DATA_BLOCK "Drives --> Plc"	// DB 1
TITLE = DRIVE --> PLC DATA BLOCK
AUTHOR : Milesi
VERSION : 0.1
  STRUCT
   TRVERSE_STATUS_W1 : STRUCT
    DB1_DBX0_0 : BOOL ;	//Setpoint/actual value deviation detected
    DB1_DBX0_1 : BOOL ;	//PZD control requests
    DB1_DBX0_2 : BOOL ;	//Actual value>=Comparsion setpoint
    DB1_DBX0_3 : BOOL ;	//Undervoltage fault
    DB1_DBX0_4 : BOOL ;	//Request to energize main contactor
    DB1_DBX0_5 : BOOL ;	//Ramp-function generetor active
    DB1_DBX0_6 : BOOL ;	//Positive speed setpoint
    DB1_DBX0_7 : BOOL ;	//Kinetic buffering/flexible response active
    DB1_DBX1_0 : BOOL ;	//Ready to switch on
    DB1_DBX1_1 : BOOL ;	//Ready to operate
    DB1_DBX1_2 : BOOL ;	//Run
    DB1_DBX1_3 : BOOL ;	//Fault is active
    DB1_DBX1_4 : BOOL ;	//OFF2 applied
    DB1_DBX1_5 : BOOL ;	//OFF3 applied
    DB1_DBX1_6 : BOOL ;	//Switch on inhibit
    DB1_DBX1_7 : BOOL ;	//Alarm is active
   END_STRUCT ;
   TRAVERSE_STATUS_W2 : STRUCT
    DB1_DBX2_0 : BOOL ;	//Power section overtemperature alarm active
    DB1_DBX2_1 : BOOL ;	//Motor overtemperature alarm active
    DB1_DBX2_2 : BOOL ;	//Motor overtemperature fault active
    DB1_DBX2_3 : BOOL ;	//Spare
    DB1_DBX2_4 : BOOL ;	//Motor locked fault active
    DB1_DBX2_5 : BOOL ;	//Spare
    DB1_DBX2_6 : BOOL ;	//Spare
    DB1_DBX2_7 : BOOL ;	//Spare
    DB1_DBX3_0 : BOOL ;	//Spare
    DB1_DBX3_1 : BOOL ;	//Spare
    DB1_DBX3_2 : BOOL ;	//Overspeed
    DB1_DBX3_3 : BOOL ;	//External fault 1 active
    DB1_DBX3_4 : BOOL ;	//External fault 2 active
    DB1_DBX3_5 : BOOL ;	//External alarm active
    DB1_DBX3_6 : BOOL ;	//Power section overload alarm active
    DB1_DBX3_7 : BOOL ;	//Power section overtemperature fault active
   END_STRUCT ;
   DB1_DBW4 : INT ;
   DB1_DBW6 : INT ;	//Motor speed
   DB1_DBW8 : INT ;	//Motor current
   DB1_DBW10 : INT ;	//Motor voltage
   DB1_DBW12 : INT ;
   DB1_DBW14 : INT ;
   DB1_DBW16 : INT ;
   DB1_DBW18 : INT ;
   DB1_DBW20 : INT ;
   DB1_DBW22 : INT ;
   DB1_DBW24 : INT ;
   DB1_DBW26 : INT ;
   DB1_DBW28 : INT ;
   DB1_DBW30 : INT ;
   DB1_DBW32 : INT ;
   DB1_DBW34 : INT ;
   DB1_DBW36 : INT ;
   DB1_DBW38 : INT ;
   BOBBIN_STATUS_W1 : STRUCT
    DB1_DBX40_0 : BOOL ;	//Setpoint/actual value deviation detected
    DB1_DBX40_1 : BOOL ;	//PZD control requests
    DB1_DBX40_2 : BOOL ;	//Actual value>=Comparsion setpoint
    DB1_DBX40_3 : BOOL ;	//Undervoltage fault
    DB1_DBX40_4 : BOOL ;	//Request to energize main contactor
    DB1_DBX40_5 : BOOL ;	//Ramp-function generetor active
    DB1_DBX40_6 : BOOL ;	//Positive speed setpoint
    DB1_DBX40_7 : BOOL ;	//Kinetic buffering/flexible response active
    DB1_DBX41_0 : BOOL ;	//Ready to switch on
    DB1_DBX41_1 : BOOL ;	//Ready to operate
    DB1_DBX41_2 : BOOL ;	//Run
    DB1_DBX41_3 : BOOL ;	//Fault is active
    DB1_DBX41_4 : BOOL ;	//OFF2 applied
    DB1_DBX41_5 : BOOL ;	//OFF3 applied
    DB1_DBX41_6 : BOOL ;	//Switch on inhibit
    DB1_DBX41_7 : BOOL ;	//Alarm is active
   END_STRUCT ;
   BOBBIN_STATUS_W2 : STRUCT
    DB1_DBX42_0 : BOOL ;	//Power section overtemperature alarm active
    DB1_DBX42_1 : BOOL ;	//Motor overtemperature alarm active
    DB1_DBX42_2 : BOOL ;	//Motor overtemperature fault active
    DB1_DBX42_3 : BOOL ;	//Spare
    DB1_DBX42_4 : BOOL ;	//Motor locked fault active
    DB1_DBX42_5 : BOOL ;	//Spare
    DB1_DBX42_6 : BOOL ;	//Spare
    DB1_DBX42_7 : BOOL ;	//Spare
    DB1_DBX43_0 : BOOL ;	//Spare
    DB1_DBX43_1 : BOOL ;	//Spare
    DB1_DBX43_2 : BOOL ;	//Overspeed
    DB1_DBX43_3 : BOOL ;	//External fault 1 active
    DB1_DBX43_4 : BOOL ;	//External fault 2 active
    DB1_DBX43_5 : BOOL ;	//External alarm active
    DB1_DBX43_6 : BOOL ;	//Power section overload alarm active
    DB1_DBX43_7 : BOOL ;	//Power section overtemperature fault active
   END_STRUCT ;
   DB1_DBW44 : INT ;
   DB1_DBW46 : INT ;	//Motor speed
   DB1_DBW48 : INT ;	//Motor current
   DB1_DBW50 : INT ;	//Motor voltage
   DB1_DBW52 : INT ;
   DB1_DBW54 : INT ;
   DB1_DBW56 : INT ;
   DB1_DBW58 : INT ;
   DB1_DBW60 : INT ;
   DB1_DBW62 : INT ;
   DB1_DBW64 : INT ;
   DB1_DBW66 : INT ;
   DB1_DBW68 : INT ;
   DB1_DBW70 : INT ;
   DB1_DBW72 : INT ;
   DB1_DBW74 : INT ;
   DB1_DBW76 : INT ;
   DB1_DBW78 : INT ;
   CAPSTAN_STATUS_W1 : STRUCT
    DB1_DBX80_0 : BOOL ;	//Setpoint/actual value deviation detected
    DB1_DBX80_1 : BOOL ;	//PZD control requests
    DB1_DBX80_2 : BOOL ;	//Actual value>=Comparsion setpoint
    DB1_DBX80_3 : BOOL ;	//Undervoltage fault
    DB1_DBX80_4 : BOOL ;	//Request to energize main contactor
    DB1_DBX80_5 : BOOL ;	//Ramp-function generetor active
    DB1_DBX80_6 : BOOL ;	//Positive speed setpoint
    DB1_DBX80_7 : BOOL ;	//Kinetic buffering/flexible response active
    DB1_DBX81_0 : BOOL ;	//Ready to switch on
    DB1_DBX81_1 : BOOL ;	//Ready to operate
    DB1_DBX81_2 : BOOL ;	//Run
    DB1_DBX81_3 : BOOL ;	//Fault is active
    DB1_DBX81_4 : BOOL ;	//OFF2 applied
    DB1_DBX81_5 : BOOL ;	//OFF3 applied
    DB1_DBX81_6 : BOOL ;	//Switch on inhibit
    DB1_DBX81_7 : BOOL ;	//Alarm is active
   END_STRUCT ;
   CAPSTAN_STATUS_W2 : STRUCT
    DB1_DBX82_0 : BOOL ;	//Power section overtemperature alarm active
    DB1_DBX82_1 : BOOL ;	//Motor overtemperature alarm active
    DB1_DBX82_2 : BOOL ;	//Motor overtemperature fault active
    DB1_DBX82_3 : BOOL ;	//Spare
    DB1_DBX82_4 : BOOL ;	//Motor locked fault active
    DB1_DBX82_5 : BOOL ;	//Spare
    DB1_DBX82_6 : BOOL ;	//Spare
    DB1_DBX82_7 : BOOL ;	//Spare
    DB1_DBX83_0 : BOOL ;	//Spare
    DB1_DBX83_1 : BOOL ;	//Spare
    DB1_DBX83_2 : BOOL ;	//Overspeed
    DB1_DBX83_3 : BOOL ;	//External fault 1 active
    DB1_DBX83_4 : BOOL ;	//External fault 2 active
    DB1_DBX83_5 : BOOL ;	//External alarm active
    DB1_DBX83_6 : BOOL ;	//Power section overload alarm active
    DB1_DBX83_7 : BOOL ;	//Power section overtemperature fault active
   END_STRUCT ;
   DB1_DBW84 : INT ;
   DB1_DBW86 : INT ;	//Motor speed
   DB1_DBW88 : INT ;	//Motor current
   DB1_DBW90 : INT ;	//Motor voltage
   DB1_DBW92 : INT ;
   DB1_DBW94 : INT ;
   DB1_DBW96 : INT ;
   DB1_DBW98 : INT ;
   DB1_DBW100 : INT ;
   DB1_DBW102 : INT ;
   DB1_DBW104 : INT ;
   DB1_DBW106 : INT ;
   DB1_DBW108 : INT ;
   DB1_DBW110 : INT ;
   DB1_DBW112 : INT ;
   DB1_DBW114 : INT ;
   DB1_DBW116 : INT ;
   DB1_DBW118 : INT ;
   CAGE_24_PREF_STATUS_W1 : STRUCT
    DB1_DBX120_0 : BOOL ;	//Setpoint/actual value deviation detected
    DB1_DBX120_1 : BOOL ;	//PZD control requests
    DB1_DBX120_2 : BOOL ;	//Actual value>=Comparsion setpoint
    DB1_DBX120_3 : BOOL ;	//Undervoltage fault
    DB1_DBX120_4 : BOOL ;	//Request to energize main contactor
    DB1_DBX120_5 : BOOL ;	//Ramp-function generetor active
    DB1_DBX120_6 : BOOL ;	//Positive speed setpoint
    DB1_DBX120_7 : BOOL ;	//Kinetic buffering/flexible response active
    DB1_DBX121_0 : BOOL ;	//Ready to switch on
    DB1_DBX121_1 : BOOL ;	//Ready to operate
    DB1_DBX121_2 : BOOL ;	//Run
    DB1_DBX121_3 : BOOL ;	//Fault is active
    DB1_DBX121_4 : BOOL ;	//OFF2 applied
    DB1_DBX121_5 : BOOL ;	//OFF3 applied
    DB1_DBX121_6 : BOOL ;	//Switch on inhibit
    DB1_DBX121_7 : BOOL ;	//Alarm is active
   END_STRUCT ;
   CAGE_24_PREF_STATUS_W2 : STRUCT
    DB1_DBX122_0 : BOOL ;	//Power section overtemperature alarm active
    DB1_DBX122_1 : BOOL ;	//Motor overtemperature alarm active
    DB1_DBX122_2 : BOOL ;	//Motor overtemperature fault active
    DB1_DBX122_3 : BOOL ;	//Spare
    DB1_DBX122_4 : BOOL ;	//Motor locked fault active
    DB1_DBX122_5 : BOOL ;	//Spare
    DB1_DBX122_6 : BOOL ;	//Spare
    DB1_DBX122_7 : BOOL ;	//Spare
    DB1_DBX123_0 : BOOL ;	//Spare
    DB1_DBX123_1 : BOOL ;	//Spare
    DB1_DBX123_2 : BOOL ;	//Overspeed
    DB1_DBX123_3 : BOOL ;	//External fault 1 active
    DB1_DBX123_4 : BOOL ;	//External fault 2 active
    DB1_DBX123_5 : BOOL ;	//External alarm active
    DB1_DBX123_6 : BOOL ;	//Power section overload alarm active
    DB1_DBX123_7 : BOOL ;	//Power section overtemperature fault active
   END_STRUCT ;
   DB1_DBW124 : INT ;
   DB1_DBW126 : INT ;	//Motor speed
   DB1_DBW128 : INT ;	//Motor current
   DB1_DBW130 : INT ;	//Motor voltage
   DB1_DBW132 : INT ;
   DB1_DBW134 : INT ;
   DB1_DBW136 : INT ;
   DB1_DBW138 : INT ;
   DB1_DBW140 : INT ;
   DB1_DBW142 : INT ;
   DB1_DBW144 : INT ;
   DB1_DBW146 : INT ;
   DB1_DBW148 : INT ;
   DB1_DBW150 : INT ;
   DB1_DBW152 : INT ;
   DB1_DBW154 : INT ;
   DB1_DBW156 : INT ;
   DB1_DBW158 : INT ;
   CAGE_24_STATUS_W1 : STRUCT
    DB1_DBX160_0 : BOOL ;	//Setpoint/actual value deviation detected
    DB1_DBX160_1 : BOOL ;	//PZD control requests
    DB1_DBX160_2 : BOOL ;	//Actual value>=Comparsion setpoint
    DB1_DBX160_3 : BOOL ;	//Undervoltage fault
    DB1_DBX160_4 : BOOL ;	//Request to energize main contactor
    DB1_DBX160_5 : BOOL ;	//Ramp-function generetor active
    DB1_DBX160_6 : BOOL ;	//Positive speed setpoint
    DB1_DBX160_7 : BOOL ;	//Kinetic buffering/flexible response active
    DB1_DBX161_0 : BOOL ;	//Ready to switch on
    DB1_DBX161_1 : BOOL ;	//Ready to operate
    DB1_DBX161_2 : BOOL ;	//Run
    DB1_DBX161_3 : BOOL ;	//Fault is active
    DB1_DBX161_4 : BOOL ;	//OFF2 applied
    DB1_DBX161_5 : BOOL ;	//OFF3 applied
    DB1_DBX161_6 : BOOL ;	//Switch on inhibit
    DB1_DBX161_7 : BOOL ;	//Alarm is active
   END_STRUCT ;
   CAGE_24_STATUS_W2 : STRUCT
    DB1_DBX162_0 : BOOL ;	//Power section overtemperature alarm active
    DB1_DBX162_1 : BOOL ;	//Motor overtemperature alarm active
    DB1_DBX162_2 : BOOL ;	//Motor overtemperature fault active
    DB1_DBX162_3 : BOOL ;	//Spare
    DB1_DBX162_4 : BOOL ;	//Motor locked fault active
    DB1_DBX162_5 : BOOL ;	//Spare
    DB1_DBX162_6 : BOOL ;	//Spare
    DB1_DBX162_7 : BOOL ;	//Spare
    DB1_DBX163_0 : BOOL ;	//Spare
    DB1_DBX163_1 : BOOL ;	//Spare
    DB1_DBX163_2 : BOOL ;	//Overspeed
    DB1_DBX163_3 : BOOL ;	//External fault 1 active
    DB1_DBX163_4 : BOOL ;	//External fault 2 active
    DB1_DBX163_5 : BOOL ;	//External alarm active
    DB1_DBX163_6 : BOOL ;	//Power section overload alarm active
    DB1_DBX163_7 : BOOL ;	//Power section overtemperature fault active
   END_STRUCT ;
   DB1_DBW1641 : INT ;
   DB1_DBW1661 : INT ;	//Motor speed
   DB1_DBW1681 : INT ;	//Motor current
   DB1_DBW1701 : INT ;	//Motor voltage
   DB1_DBW1721 : INT ;
   DB1_DBW1741 : INT ;
   DB1_DBW1761 : INT ;
   DB1_DBW1781 : INT ;
   DB1_DBW1801 : INT ;
   DB1_DBW1821 : INT ;
   DB1_DBW1841 : INT ;
   DB1_DBW1861 : INT ;
   DB1_DBW1881 : INT ;
   DB1_DBW1901 : INT ;
   DB1_DBW1921 : INT ;
   DB1_DBW1941 : INT ;
   DB1_DBW1961 : INT ;
   DB1_DBW1981 : INT ;
   CAGE_18_PREF_STATUS_W1 : STRUCT
    DB1_DBX200_0 : BOOL ;	//Setpoint/actual value deviation detected
    DB1_DBX200_1 : BOOL ;	//PZD control requests
    DB1_DBX200_2 : BOOL ;	//Actual value>=Comparsion setpoint
    DB1_DBX200_3 : BOOL ;	//Undervoltage fault
    DB1_DBX200_4 : BOOL ;	//Request to energize main contactor
    DB1_DBX200_5 : BOOL ;	//Ramp-function generetor active
    DB1_DBX200_6 : BOOL ;	//Positive speed setpoint
    DB1_DBX200_7 : BOOL ;	//Kinetic buffering/flexible response active
    DB1_DBX201_0 : BOOL ;	//Ready to switch on
    DB1_DBX201_1 : BOOL ;	//Ready to operate
    DB1_DBX201_2 : BOOL ;	//Run
    DB1_DBX201_3 : BOOL ;	//Fault is active
    DB1_DBX201_4 : BOOL ;	//OFF2 applied
    DB1_DBX201_5 : BOOL ;	//OFF3 applied
    DB1_DBX201_6 : BOOL ;	//Switch on inhibit
    DB1_DBX201_7 : BOOL ;	//Alarm is active
   END_STRUCT ;
   CAGE_18_PREF_STATUS_W2 : STRUCT
    DB1_DBX202_0 : BOOL ;	//Power section overtemperature alarm active
    DB1_DBX202_1 : BOOL ;	//Motor overtemperature alarm active
    DB1_DBX202_2 : BOOL ;	//Motor overtemperature fault active
    DB1_DBX202_3 : BOOL ;	//Spare
    DB1_DBX202_4 : BOOL ;	//Motor locked fault active
    DB1_DBX202_5 : BOOL ;	//Spare
    DB1_DBX202_6 : BOOL ;	//Spare
    DB1_DBX202_7 : BOOL ;	//Spare
    DB1_DBX203_0 : BOOL ;	//Spare
    DB1_DBX203_1 : BOOL ;	//Spare
    DB1_DBX203_2 : BOOL ;	//Overspeed
    DB1_DBX203_3 : BOOL ;	//External fault 1 active
    DB1_DBX203_4 : BOOL ;	//External fault 2 active
    DB1_DBX203_5 : BOOL ;	//External alarm active
    DB1_DBX203_6 : BOOL ;	//Power section overload alarm active
    DB1_DBX203_7 : BOOL ;	//Power section overtemperature fault active
   END_STRUCT ;
   DB1_DBW204 : INT ;
   DB1_DBW206 : INT ;	//Motor speed
   DB1_DBW208 : INT ;	//Motor current
   DB1_DBW210 : INT ;	//Motor voltage
   DB1_DBW212 : INT ;
   DB1_DBW214 : INT ;
   DB1_DBW216 : INT ;
   DB1_DBW218 : INT ;
   DB1_DBW220 : INT ;
   DB1_DBW222 : INT ;
   DB1_DBW224 : INT ;
   DB1_DBW226 : INT ;
   DB1_DBW228 : INT ;
   DB1_DBW230 : INT ;
   DB1_DBW232 : INT ;
   DB1_DBW234 : INT ;
   DB1_DBW236 : INT ;
   DB1_DBW238 : INT ;
   CAGE_18_STATUS_W1 : STRUCT
    DB1_DBX240_0 : BOOL ;	//Setpoint/actual value deviation detected
    DB1_DBX240_1 : BOOL ;	//PZD control requests
    DB1_DBX240_2 : BOOL ;	//Actual value>=Comparsion setpoint
    DB1_DBX240_3 : BOOL ;	//Undervoltage fault
    DB1_DBX240_4 : BOOL ;	//Request to energize main contactor
    DB1_DBX240_5 : BOOL ;	//Ramp-function generetor active
    DB1_DBX240_6 : BOOL ;	//Positive speed setpoint
    DB1_DBX240_7 : BOOL ;	//Kinetic buffering/flexible response active
    DB1_DBX241_0 : BOOL ;	//Ready to switch on
    DB1_DBX241_1 : BOOL ;	//Ready to operate
    DB1_DBX241_2 : BOOL ;	//Run
    DB1_DBX241_3 : BOOL ;	//Fault is active
    DB1_DBX241_4 : BOOL ;	//OFF2 applied
    DB1_DBX241_5 : BOOL ;	//OFF3 applied
    DB1_DBX241_6 : BOOL ;	//Switch on inhibit
    DB1_DBX241_7 : BOOL ;	//Alarm is active
   END_STRUCT ;
   CAGE_18_STATUS_W2 : STRUCT
    DB1_DBX242_0 : BOOL ;	//Power section overtemperature alarm active
    DB1_DBX242_1 : BOOL ;	//Motor overtemperature alarm active
    DB1_DBX242_2 : BOOL ;	//Motor overtemperature fault active
    DB1_DBX242_3 : BOOL ;	//Spare
    DB1_DBX242_4 : BOOL ;	//Motor locked fault active
    DB1_DBX242_5 : BOOL ;	//Spare
    DB1_DBX242_6 : BOOL ;	//Spare
    DB1_DBX242_7 : BOOL ;	//Spare
    DB1_DBX243_0 : BOOL ;	//Spare
    DB1_DBX243_1 : BOOL ;	//Spare
    DB1_DBX243_2 : BOOL ;	//Overspeed
    DB1_DBX243_3 : BOOL ;	//External fault 1 active
    DB1_DBX243_4 : BOOL ;	//External fault 2 active
    DB1_DBX243_5 : BOOL ;	//External alarm active
    DB1_DBX243_6 : BOOL ;	//Power section overload alarm active
    DB1_DBX243_7 : BOOL ;	//Power section overtemperature fault active
   END_STRUCT ;
   DB1_DBW244 : INT ;
   DB1_DBW246 : INT ;	//Motor speed
   DB1_DBW248 : INT ;	//Motor current
   DB1_DBW250 : INT ;	//Motor voltage
   DB1_DBW252 : INT ;
   DB1_DBW254 : INT ;
   DB1_DBW256 : INT ;
   DB1_DBW258 : INT ;
   DB1_DBW260 : INT ;
   DB1_DBW262 : INT ;
   DB1_DBW264 : INT ;
   DB1_DBW266 : INT ;
   DB1_DBW268 : INT ;
   DB1_DBW270 : INT ;
   DB1_DBW272 : INT ;
   DB1_DBW274 : INT ;
   DB1_DBW276 : INT ;
   DB1_DBW278 : INT ;
   CAGE_12_PREF_STATUS_W1 : STRUCT
    DB1_DBX280_0 : BOOL ;	//Setpoint/actual value deviation detected
    DB1_DBX280_1 : BOOL ;	//PZD control requests
    DB1_DBX280_2 : BOOL ;	//Actual value>=Comparsion setpoint
    DB1_DBX280_3 : BOOL ;	//Undervoltage fault
    DB1_DBX280_4 : BOOL ;	//Request to energize main contactor
    DB1_DBX280_5 : BOOL ;	//Ramp-function generetor active
    DB1_DBX280_6 : BOOL ;	//Positive speed setpoint
    DB1_DBX280_7 : BOOL ;	//Kinetic buffering/flexible response active
    DB1_DBX281_0 : BOOL ;	//Ready to switch on
    DB1_DBX281_1 : BOOL ;	//Ready to operate
    DB1_DBX281_2 : BOOL ;	//Run
    DB1_DBX281_3 : BOOL ;	//Fault is active
    DB1_DBX281_4 : BOOL ;	//OFF2 applied
    DB1_DBX281_5 : BOOL ;	//OFF3 applied
    DB1_DBX281_6 : BOOL ;	//Switch on inhibit
    DB1_DBX281_7 : BOOL ;	//Alarm is active
   END_STRUCT ;
   CAGE_12_PREF_STATUS_W2 : STRUCT
    DB1_DBX282_0 : BOOL ;	//Power section overtemperature alarm active
    DB1_DBX282_1 : BOOL ;	//Motor overtemperature alarm active
    DB1_DBX282_2 : BOOL ;	//Motor overtemperature fault active
    DB1_DBX282_3 : BOOL ;	//Spare
    DB1_DBX282_4 : BOOL ;	//Motor locked fault active
    DB1_DBX282_5 : BOOL ;	//Spare
    DB1_DBX282_6 : BOOL ;	//Spare
    DB1_DBX282_7 : BOOL ;	//Spare
    DB1_DBX283_0 : BOOL ;	//Spare
    DB1_DBX283_1 : BOOL ;	//Spare
    DB1_DBX283_2 : BOOL ;	//Overspeed
    DB1_DBX283_3 : BOOL ;	//External fault 1 active
    DB1_DBX283_4 : BOOL ;	//External fault 2 active
    DB1_DBX283_5 : BOOL ;	//External alarm active
    DB1_DBX283_6 : BOOL ;	//Power section overload alarm active
    DB1_DBX283_7 : BOOL ;	//Power section overtemperature fault active
   END_STRUCT ;
   DB1_DBW284 : INT ;
   DB1_DBW286 : INT ;	//Motor speed
   DB1_DBW288 : INT ;	//Motor current
   DB1_DBW290 : INT ;	//Motor voltage
   DB1_DBW292 : INT ;
   DB1_DBW294 : INT ;
   DB1_DBW296 : INT ;
   DB1_DBW298 : INT ;
   DB1_DBW300 : INT ;
   DB1_DBW302 : INT ;
   DB1_DBW304 : INT ;
   DB1_DBW306 : INT ;
   DB1_DBW308 : INT ;
   DB1_DBW310 : INT ;
   DB1_DBW312 : INT ;
   DB1_DBW314 : INT ;
   DB1_DBW316 : INT ;
   DB1_DBW318 : INT ;
   CAGE_12_STATUS_W1 : STRUCT
    DB1_DBX320_0 : BOOL ;	//Setpoint/actual value deviation detected
    DB1_DBX320_1 : BOOL ;	//PZD control requests
    DB1_DBX320_2 : BOOL ;	//Actual value>=Comparsion setpoint
    DB1_DBX320_3 : BOOL ;	//Undervoltage fault
    DB1_DBX320_4 : BOOL ;	//Request to energize main contactor
    DB1_DBX320_5 : BOOL ;	//Ramp-function generetor active
    DB1_DBX320_6 : BOOL ;	//Positive speed setpoint
    DB1_DBX320_7 : BOOL ;	//Kinetic buffering/flexible response active
    DB1_DBX321_0 : BOOL ;	//Ready to switch on
    DB1_DBX321_1 : BOOL ;	//Ready to operate
    DB1_DBX321_2 : BOOL ;	//Run
    DB1_DBX321_3 : BOOL ;	//Fault is active
    DB1_DBX321_4 : BOOL ;	//OFF2 applied
    DB1_DBX321_5 : BOOL ;	//OFF3 applied
    DB1_DBX321_6 : BOOL ;	//Switch on inhibit
    DB1_DBX321_7 : BOOL ;	//Alarm is active
   END_STRUCT ;
   CAGE_12_STATUS_W2 : STRUCT
    DB1_DBX322_0 : BOOL ;	//Power section overtemperature alarm active
    DB1_DBX322_1 : BOOL ;	//Motor overtemperature alarm active
    DB1_DBX322_2 : BOOL ;	//Motor overtemperature fault active
    DB1_DBX322_3 : BOOL ;	//Spare
    DB1_DBX322_4 : BOOL ;	//Motor locked fault active
    DB1_DBX322_5 : BOOL ;	//Spare
    DB1_DBX322_6 : BOOL ;	//Spare
    DB1_DBX322_7 : BOOL ;	//Spare
    DB1_DBX323_0 : BOOL ;	//Spare
    DB1_DBX323_1 : BOOL ;	//Spare
    DB1_DBX323_2 : BOOL ;	//Overspeed
    DB1_DBX323_3 : BOOL ;	//External fault 1 active
    DB1_DBX323_4 : BOOL ;	//External fault 2 active
    DB1_DBX323_5 : BOOL ;	//External alarm active
    DB1_DBX323_6 : BOOL ;	//Power section overload alarm active
    DB1_DBX323_7 : BOOL ;	//Power section overtemperature fault active
   END_STRUCT ;
   DB1_DBW324 : INT ;
   DB1_DBW326 : INT ;	//Motor speed
   DB1_DBW328 : INT ;	//Motor current
   DB1_DBW330 : INT ;	//Motor voltage
   DB1_DBW332 : INT ;
   DB1_DBW334 : INT ;
   DB1_DBW336 : INT ;
   DB1_DBW338 : INT ;
   DB1_DBW340 : INT ;
   DB1_DBW342 : INT ;
   DB1_DBW344 : INT ;
   DB1_DBW346 : INT ;
   DB1_DBW348 : INT ;
   DB1_DBW350 : INT ;
   DB1_DBW352 : INT ;
   DB1_DBW354 : INT ;
   DB1_DBW356 : INT ;
   DB1_DBW358 : INT ;
   CAGE_6_STATUS_W1 : STRUCT
    DB1_DBX360_0 : BOOL ;	//Setpoint/actual value deviation detected
    DB1_DBX360_1 : BOOL ;	//PZD control requests
    DB1_DBX360_2 : BOOL ;	//Actual value>=Comparsion setpoint
    DB1_DBX360_3 : BOOL ;	//Undervoltage fault
    DB1_DBX360_4 : BOOL ;	//Request to energize main contactor
    DB1_DBX360_5 : BOOL ;	//Ramp-function generetor active
    DB1_DBX360_6 : BOOL ;	//Positive speed setpoint
    DB1_DBX360_7 : BOOL ;	//Kinetic buffering/flexible response active
    DB1_DBX361_0 : BOOL ;	//Ready to switch on
    DB1_DBX361_1 : BOOL ;	//Ready to operate
    DB1_DBX361_2 : BOOL ;	//Run
    DB1_DBX361_3 : BOOL ;	//Fault is active
    DB1_DBX361_4 : BOOL ;	//OFF2 applied
    DB1_DBX361_5 : BOOL ;	//OFF3 applied
    DB1_DBX361_6 : BOOL ;	//Switch on inhibit
    DB1_DBX361_7 : BOOL ;	//Alarm is active
   END_STRUCT ;
   CAGE_6_STATUS_W2 : STRUCT
    DB1_DBX362_0 : BOOL ;	//Power section overtemperature alarm active
    DB1_DBX362_1 : BOOL ;	//Motor overtemperature alarm active
    DB1_DBX362_2 : BOOL ;	//Motor overtemperature fault active
    DB1_DBX362_3 : BOOL ;	//Spare
    DB1_DBX362_4 : BOOL ;	//Motor locked fault active
    DB1_DBX362_5 : BOOL ;	//Spare
    DB1_DBX362_6 : BOOL ;	//Spare
    DB1_DBX362_7 : BOOL ;	//Spare
    DB1_DBX363_0 : BOOL ;	//Spare
    DB1_DBX363_1 : BOOL ;	//Spare
    DB1_DBX363_2 : BOOL ;	//Overspeed
    DB1_DBX363_3 : BOOL ;	//External fault 1 active
    DB1_DBX363_4 : BOOL ;	//External fault 2 active
    DB1_DBX363_5 : BOOL ;	//External alarm active
    DB1_DBX363_6 : BOOL ;	//Power section overload alarm active
    DB1_DBX363_7 : BOOL ;	//Power section overtemperature fault active
   END_STRUCT ;
   DB1_DBW364 : INT ;
   DB1_DBW366 : INT ;	//Motor speed
   DB1_DBW368 : INT ;	//Motor current
   DB1_DBW370 : INT ;	//Motor voltage
   DB1_DBW372 : INT ;
   DB1_DBW374 : INT ;
   DB1_DBW376 : INT ;
   DB1_DBW378 : INT ;
   DB1_DBW380 : INT ;
   DB1_DBW382 : INT ;
   DB1_DBW384 : INT ;
   DB1_DBW386 : INT ;
   DB1_DBW388 : INT ;
   DB1_DBW390 : INT ;
   DB1_DBW392 : INT ;
   DB1_DBW394 : INT ;
   DB1_DBW396 : INT ;
   DB1_DBW398 : INT ;
   SPARE_STATUS_W1 : STRUCT
    DB1_DBX400_0 : BOOL ;	//Setpoint/actual value deviation detected
    DB1_DBX400_1 : BOOL ;	//PZD control requests
    DB1_DBX400_2 : BOOL ;	//Actual value>=Comparsion setpoint
    DB1_DBX400_3 : BOOL ;	//Undervoltage fault
    DB1_DBX400_4 : BOOL ;	//Request to energize main contactor
    DB1_DBX400_5 : BOOL ;	//Ramp-function generetor active
    DB1_DBX400_6 : BOOL ;	//Positive speed setpoint
    DB1_DBX400_7 : BOOL ;	//Kinetic buffering/flexible response active
    DB1_DBX401_0 : BOOL ;	//Ready to switch on
    DB1_DBX401_1 : BOOL ;	//Ready to operate
    DB1_DBX401_2 : BOOL ;	//Run
    DB1_DBX401_3 : BOOL ;	//Fault is active
    DB1_DBX401_4 : BOOL ;	//OFF2 applied
    DB1_DBX401_5 : BOOL ;	//OFF3 applied
    DB1_DBX401_6 : BOOL ;	//Switch on inhibit
    DB1_DBX401_7 : BOOL ;	//Alarm is active
   END_STRUCT ;
   SPARE_STATUS_W2 : STRUCT
    DB1_DBX402_0 : BOOL ;	//Power section overtemperature alarm active
    DB1_DBX402_1 : BOOL ;	//Motor overtemperature alarm active
    DB1_DBX402_2 : BOOL ;	//Motor overtemperature fault active
    DB1_DBX402_3 : BOOL ;	//Spare
    DB1_DBX402_4 : BOOL ;	//Motor locked fault active
    DB1_DBX402_5 : BOOL ;	//Spare
    DB1_DBX402_6 : BOOL ;	//Spare
    DB1_DBX402_7 : BOOL ;	//Spare
    DB1_DBX403_0 : BOOL ;	//Spare
    DB1_DBX403_1 : BOOL ;	//Spare
    DB1_DBX403_2 : BOOL ;	//Overspeed
    DB1_DBX403_3 : BOOL ;	//External fault 1 active
    DB1_DBX403_4 : BOOL ;	//External fault 2 active
    DB1_DBX403_5 : BOOL ;	//External alarm active
    DB1_DBX403_6 : BOOL ;	//Power section overload alarm active
    DB1_DBX403_7 : BOOL ;	//Power section overtemperature fault active
   END_STRUCT ;
   DB1_DBW404 : INT ;
   DB2_DBW406 : INT ;
   DB2_DBW408 : INT ;
   DB2_DBW410 : INT ;
   DB2_DBW412 : INT ;
   DB2_DBW414 : INT ;
   DB2_DBW416 : INT ;
   DB2_DBW418 : INT ;
   DB2_DBW420 : INT ;
   DB2_DBW422 : INT ;
   DB2_DBW424 : INT ;
   DB2_DBW426 : INT ;
   DB2_DBW428 : INT ;
   DB2_DBW430 : INT ;
   DB2_DBW432 : INT ;
   DB2_DBW434 : INT ;
   DB2_DBW436 : INT ;
   DB2_DBW438 : INT ;
   DB2_DBW440 : INT ;
   DB2_DBW442 : INT ;
   DB2_DBW444 : INT ;
   DB2_DBW446 : INT ;
   DB2_DBW448 : INT ;
   DB2_DBW450 : INT ;
   DB2_DBW452 : INT ;
   DB2_DBW454 : INT ;
   DB2_DBW456 : INT ;
   DB2_DBW458 : INT ;
   DB2_DBW460 : INT ;
   DB2_DBW462 : INT ;
   DB2_DBW464 : INT ;
   DB2_DBW466 : INT ;
   DB2_DBW468 : INT ;
   DB2_DBW470 : INT ;
   DB2_DBW472 : INT ;
   DB2_DBW474 : INT ;
   DB2_DBW476 : INT ;
   DB2_DBW478 : INT ;
   DB2_DBW480 : INT ;
   DB2_DBW482 : INT ;
   DB2_DBW484 : INT ;
   DB2_DBW486 : INT ;
   DB2_DBW488 : INT ;
   DB2_DBW490 : INT ;
   DB2_DBW492 : INT ;
   DB2_DBW494 : INT ;
   DB2_DBW496 : INT ;
   DB2_DBW498 : INT ;
   PKW_READ_CAGE24 : STRUCT
    DB1_DBW500 : INT ;	//PKE
    DB1_DBW502 : INT ;	//IND
    DB1_DBW504 : INT ;	//PWE1
    DB1_DBW506 : INT ;	//PWE2
   END_STRUCT ;
   DB1_DBW508 : INT ;	//Spare
   PKW_READ_CAGE18 : STRUCT
    DB1_DBW510 : INT ;	//PKE
    DB1_DBW512 : INT ;	//IND
    DB1_DBW514 : INT ;	//PWE1
    DB1_DBW516 : INT ;	//PWE2
   END_STRUCT ;
   DB1_DBW518 : INT ;	//Spare
   PKW_READ_CAGE12 : STRUCT
    DB1_DBW520 : INT ;	//PKE
    DB1_DBW522 : INT ;	//IND
    DB1_DBW524 : INT ;	//PWE1
    DB1_DBW526 : INT ;	//PWE2
   END_STRUCT ;
   DB1_DBW528 : INT ;	//Spare
   PKW_READ_CAGE6 : STRUCT
    DB1_DBW530 : INT ;	//PKE
    DB1_DBW532 : INT ;	//IND
    DB1_DBW534 : INT ;	//PWE1
    DB1_DBW536 : INT ;	//PWE2
   END_STRUCT ;
   DB1_DBW538 : INT ;	//Spare
  END_STRUCT ;	
BEGIN
   TRVERSE_STATUS_W1.DB1_DBX0_0 := TRUE;
   TRVERSE_STATUS_W1.DB1_DBX0_1 := TRUE;
   TRVERSE_STATUS_W1.DB1_DBX0_6 := TRUE;
   TRVERSE_STATUS_W1.DB1_DBX1_0 := TRUE;
   TRVERSE_STATUS_W1.DB1_DBX1_4 := TRUE;
   TRVERSE_STATUS_W1.DB1_DBX1_5 := TRUE;
   TRAVERSE_STATUS_W2.DB1_DBX3_2 := TRUE;
   BOBBIN_STATUS_W1.DB1_DBX40_0 := TRUE;
   BOBBIN_STATUS_W1.DB1_DBX40_1 := TRUE;
   BOBBIN_STATUS_W1.DB1_DBX40_4 := TRUE;
   BOBBIN_STATUS_W1.DB1_DBX40_6 := TRUE;
   BOBBIN_STATUS_W1.DB1_DBX41_2 := TRUE;
   BOBBIN_STATUS_W1.DB1_DBX41_4 := TRUE;
   BOBBIN_STATUS_W1.DB1_DBX41_5 := TRUE;
   BOBBIN_STATUS_W2.DB1_DBX42_5 := TRUE;
   BOBBIN_STATUS_W2.DB1_DBX43_2 := TRUE;
   DB1_DBW48 := 2088;
   DB1_DBW50 := 524;
   CAPSTAN_STATUS_W1.DB1_DBX80_0 := TRUE;
   CAPSTAN_STATUS_W1.DB1_DBX80_1 := TRUE;
   CAPSTAN_STATUS_W1.DB1_DBX80_6 := TRUE;
   CAPSTAN_STATUS_W1.DB1_DBX81_0 := TRUE;
   CAPSTAN_STATUS_W1.DB1_DBX81_4 := TRUE;
   CAPSTAN_STATUS_W1.DB1_DBX81_5 := TRUE;
   CAPSTAN_STATUS_W2.DB1_DBX82_5 := TRUE;
   CAPSTAN_STATUS_W2.DB1_DBX83_2 := TRUE;
   CAGE_24_PREF_STATUS_W1.DB1_DBX120_0 := TRUE;
   CAGE_24_PREF_STATUS_W1.DB1_DBX120_1 := TRUE;
   CAGE_24_PREF_STATUS_W1.DB1_DBX120_6 := TRUE;
   CAGE_24_PREF_STATUS_W1.DB1_DBX121_0 := TRUE;
   CAGE_24_PREF_STATUS_W1.DB1_DBX121_4 := TRUE;
   CAGE_24_PREF_STATUS_W1.DB1_DBX121_5 := TRUE;
   CAGE_24_PREF_STATUS_W2.DB1_DBX123_2 := TRUE;
   CAGE_24_STATUS_W1.DB1_DBX160_0 := TRUE;
   CAGE_24_STATUS_W1.DB1_DBX160_1 := TRUE;
   CAGE_24_STATUS_W1.DB1_DBX160_6 := TRUE;
   CAGE_24_STATUS_W1.DB1_DBX161_0 := TRUE;
   CAGE_24_STATUS_W1.DB1_DBX161_4 := TRUE;
   CAGE_24_STATUS_W1.DB1_DBX161_5 := TRUE;
   CAGE_24_STATUS_W2.DB1_DBX163_2 := TRUE;
   CAGE_18_PREF_STATUS_W1.DB1_DBX200_0 := TRUE;
   CAGE_18_PREF_STATUS_W1.DB1_DBX200_1 := TRUE;
   CAGE_18_PREF_STATUS_W1.DB1_DBX200_6 := TRUE;
   CAGE_18_PREF_STATUS_W1.DB1_DBX201_0 := TRUE;
   CAGE_18_PREF_STATUS_W1.DB1_DBX201_4 := TRUE;
   CAGE_18_PREF_STATUS_W1.DB1_DBX201_5 := TRUE;
   CAGE_18_PREF_STATUS_W2.DB1_DBX203_2 := TRUE;
   CAGE_18_STATUS_W1.DB1_DBX240_0 := TRUE;
   CAGE_18_STATUS_W1.DB1_DBX240_1 := TRUE;
   CAGE_18_STATUS_W1.DB1_DBX240_6 := TRUE;
   CAGE_18_STATUS_W1.DB1_DBX241_0 := TRUE;
   CAGE_18_STATUS_W1.DB1_DBX241_4 := TRUE;
   CAGE_18_STATUS_W1.DB1_DBX241_5 := TRUE;
   CAGE_18_STATUS_W2.DB1_DBX243_2 := TRUE;
   CAGE_12_PREF_STATUS_W1.DB1_DBX280_0 := TRUE;
   CAGE_12_PREF_STATUS_W1.DB1_DBX280_1 := TRUE;
   CAGE_12_PREF_STATUS_W1.DB1_DBX280_6 := TRUE;
   CAGE_12_PREF_STATUS_W1.DB1_DBX281_0 := TRUE;
   CAGE_12_PREF_STATUS_W1.DB1_DBX281_4 := TRUE;
   CAGE_12_PREF_STATUS_W1.DB1_DBX281_5 := TRUE;
   CAGE_12_PREF_STATUS_W2.DB1_DBX283_2 := TRUE;
   CAGE_12_STATUS_W1.DB1_DBX320_0 := TRUE;
   CAGE_12_STATUS_W1.DB1_DBX320_1 := TRUE;
   CAGE_12_STATUS_W1.DB1_DBX320_6 := TRUE;
   CAGE_12_STATUS_W1.DB1_DBX321_0 := TRUE;
   CAGE_12_STATUS_W1.DB1_DBX321_4 := TRUE;
   CAGE_12_STATUS_W1.DB1_DBX321_5 := TRUE;
   CAGE_12_STATUS_W2.DB1_DBX322_5 := TRUE;
   CAGE_12_STATUS_W2.DB1_DBX323_2 := TRUE;
   CAGE_6_STATUS_W1.DB1_DBX360_0 := TRUE;
   CAGE_6_STATUS_W1.DB1_DBX360_1 := TRUE;
   CAGE_6_STATUS_W1.DB1_DBX360_6 := TRUE;
   CAGE_6_STATUS_W1.DB1_DBX361_0 := TRUE;
   CAGE_6_STATUS_W1.DB1_DBX361_4 := TRUE;
   CAGE_6_STATUS_W1.DB1_DBX361_5 := TRUE;
   CAGE_6_STATUS_W2.DB1_DBX362_5 := TRUE;
   CAGE_6_STATUS_W2.DB1_DBX363_2 := TRUE;
   SPARE_STATUS_W1.DB1_DBX400_0 := TRUE;
   SPARE_STATUS_W1.DB1_DBX400_1 := TRUE;
   SPARE_STATUS_W1.DB1_DBX400_6 := TRUE;
   SPARE_STATUS_W1.DB1_DBX401_0 := TRUE;
   SPARE_STATUS_W1.DB1_DBX401_4 := TRUE;
   SPARE_STATUS_W1.DB1_DBX401_5 := TRUE;
   SPARE_STATUS_W2.DB1_DBX403_2 := TRUE;
   DB1_DBW404 := 444;
   PKW_READ_CAGE24.DB1_DBW500 := 4613;
   PKW_READ_CAGE18.DB1_DBW510 := 4613;
   PKW_READ_CAGE6.DB1_DBW530 := 4613;
END_DATA_BLOCK

DATA_BLOCK "Plc --> Drives"	// DB 2
TITLE = PLC --> DRIVE DATA BLOCK
AUTHOR : Milesi
VERSION : 0.1
  STRUCT
   TRAVERSE_CONTROL_W1 : STRUCT
    DB2_DBX0_0 : BOOL ;	//Inching bit0
    DB2_DBX0_1 : BOOL ;	//Inching bit1
    DB2_DBX0_2 : BOOL ;	//Control requested
    DB2_DBX0_3 : BOOL ;	//Enable positive direction of rotation
    DB2_DBX0_4 : BOOL ;	//Enable negative direction of rotation
    DB2_DBX0_5 : BOOL ;	//Increase motorized potenziometer
    DB2_DBX0_6 : BOOL ;	//Decrease motorized potenziometer
    DB2_DBX0_7 : BOOL ;	//External fault1
    DB2_DBX1_0 : BOOL ;	//Off1
    DB2_DBX1_1 : BOOL ;	//Off2
    DB2_DBX1_2 : BOOL ;	//Off3
    DB2_DBX1_3 : BOOL ;	//Enable
    DB2_DBX1_4 : BOOL ;	//Enable ramp-function generetor
    DB2_DBX1_5 : BOOL ;	//Ramp-function generetor start
    DB2_DBX1_6 : BOOL ;	//Enable setpoint
    DB2_DBX1_7 : BOOL ;	//1Edge acknowledge
   END_STRUCT ;
   TRAVERSE_CONTROL_W2 : STRUCT
    DB2_DBX2_0 : BOOL ;	//Enable speed controller droop
    DB2_DBX2_1 : BOOL ;	//Enable speed controller
    DB2_DBX2_2 : BOOL ;	//External fault2
    DB2_DBX2_3 : BOOL ;	//Master drive
    DB2_DBX2_4 : BOOL ;	//External alarm1
    DB2_DBX2_5 : BOOL ;	//External alarm2
    DB2_DBX2_6 : BOOL ;	//Select bico data set1
    DB2_DBX2_7 : BOOL ;	//Main contactor check-back signal
    DB2_DBX3_0 : BOOL ;	//Select function data set bit0
    DB2_DBX3_1 : BOOL ;	//Select function data set bit1
    DB2_DBX3_2 : BOOL ;	//Spare
    DB2_DBX3_3 : BOOL ;	//Spare
    DB2_DBX3_4 : BOOL ;	//Select fixed setpoint0
    DB2_DBX3_5 : BOOL ;	//Select fixed setpoint1
    DB2_DBX3_6 : BOOL ;	//Spare
    DB2_DBX3_7 : BOOL ;	//Spare
   END_STRUCT ;
   DB2_DBW4 : INT ;	//Motor speed reference
   DB2_DBW6 : INT ;
   DB2_DBW8 : INT ;
   DB2_DBW10 : INT ;
   DB2_DBW12 : INT ;
   DB2_DBW14 : INT ;
   DB2_DBW16 : INT ;
   DB2_DBW18 : INT ;
   DB2_DBW20 : INT ;
   DB2_DBW22 : INT ;
   DB2_DBW24 : INT ;
   DB2_DBW26 : INT ;
   DB2_DBW28 : INT ;
   DB2_DBW30 : INT ;
   DB2_DBW32 : INT ;
   DB2_DBW34 : INT ;
   DB2_DBW36 : INT ;
   DB2_DBW38 : INT ;
   BOBBIN_CONTROL_W1 : STRUCT
    DB2_DBX40_0 : BOOL ;	//Inching bit0
    DB2_DBX40_1 : BOOL ;	//Inching bit1
    DB2_DBX40_2 : BOOL ;	//Control requested
    DB2_DBX40_3 : BOOL ;	//Enable positive direction of rotation
    DB2_DBX40_4 : BOOL ;	//Enable negative direction of rotation
    DB2_DBX40_5 : BOOL ;	//Increase motorized potenziometer
    DB2_DBX40_6 : BOOL ;	//Decrease motorized potenziometer
    DB2_DBX40_7 : BOOL ;	//External fault1
    DB2_DBX41_0 : BOOL ;	//Off1
    DB2_DBX41_1 : BOOL ;	//Off2
    DB2_DBX41_2 : BOOL ;	//Off3
    DB2_DBX41_3 : BOOL ;	//Enable
    DB2_DBX41_4 : BOOL ;	//Enable ramp-function generetor
    DB2_DBX41_5 : BOOL ;	//Ramp-function generetor start
    DB2_DBX41_6 : BOOL ;	//Enable setpoint
    DB2_DBX41_7 : BOOL ;	//1Edge acknowledge
   END_STRUCT ;
   BOBBIN_CONTROL_W2 : STRUCT
    DB2_DBX42_0 : BOOL ;	//Enable speed controller droop
    DB2_DBX42_1 : BOOL ;	//Enable speed controller
    DB2_DBX42_2 : BOOL ;	//External fault2
    DB2_DBX42_3 : BOOL ;	//Master drive
    DB2_DBX42_4 : BOOL ;	//External alarm1
    DB2_DBX42_5 : BOOL ;	//External alarm2
    DB2_DBX42_6 : BOOL ;	//Select bico data set1
    DB2_DBX42_7 : BOOL ;	//Main contactor check-back signal
    DB2_DBX43_0 : BOOL ;	//Select function data set bit0
    DB2_DBX43_1 : BOOL ;	//Select function data set bit1
    DB2_DBX43_2 : BOOL ;	//Spare
    DB2_DBX43_3 : BOOL ;	//Spare
    DB2_DBX43_4 : BOOL ;	//Select fixed setpoint0
    DB2_DBX43_5 : BOOL ;	//Select fixed setpoint1
    DB2_DBX43_6 : BOOL ;	//Spare
    DB2_DBX43_7 : BOOL ;	//Spare
   END_STRUCT ;
   DB2_DBW44 : INT ;	//Motor speed reference
   DB2_DBW46 : INT ;	//Motor pull reference
   DB2_DBW48 : INT ;
   DB2_DBW50 : INT ;
   DB2_DBW52 : INT ;
   DB2_DBW54 : INT ;
   DB2_DBW56 : INT ;
   DB2_DBW58 : INT ;
   DB2_DBW60 : INT ;
   DB2_DBW62 : INT ;
   DB2_DBW64 : INT ;
   DB2_DBW66 : INT ;
   DB2_DBW68 : INT ;
   DB2_DBW70 : INT ;
   DB2_DBW72 : INT ;
   DB2_DBW74 : INT ;
   DB2_DBW76 : INT ;
   DB2_DBW78 : INT ;
   CAPSTAN_CONTROL_W1 : STRUCT
    DB2_DBX80_0 : BOOL ;	//Inching bit0
    DB2_DBX80_1 : BOOL ;	//Inching bit1
    DB2_DBX80_2 : BOOL ;	//Control requested
    DB2_DBX80_3 : BOOL ;	//Enable positive direction of rotation
    DB2_DBX80_4 : BOOL ;	//Enable negative direction of rotation
    DB2_DBX80_5 : BOOL ;	//Increase motorized potenziometer
    DB2_DBX80_6 : BOOL ;	//Decrease motorized potenziometer
    DB2_DBX80_7 : BOOL ;	//External fault1
    DB2_DBX81_0 : BOOL ;	//Off1
    DB2_DBX81_1 : BOOL ;	//Off2
    DB2_DBX81_2 : BOOL ;	//Off3
    DB2_DBX81_3 : BOOL ;	//Enable
    DB2_DBX81_4 : BOOL ;	//Enable ramp-function generetor
    DB2_DBX81_5 : BOOL ;	//Ramp-function generetor start
    DB2_DBX81_6 : BOOL ;	//Enable setpoint
    DB2_DBX81_7 : BOOL ;	//1Edge acknowledge
   END_STRUCT ;
   CAPSTAN_CONTROL_W2 : STRUCT
    DB2_DBX82_0 : BOOL ;	//Enable speed controller droop
    DB2_DBX82_1 : BOOL ;	//Enable speed controller
    DB2_DBX82_2 : BOOL ;	//External fault2
    DB2_DBX82_3 : BOOL ;	//Master drive
    DB2_DBX82_4 : BOOL ;	//External alarm1
    DB2_DBX82_5 : BOOL ;	//External alarm2
    DB2_DBX82_6 : BOOL ;	//Select bico data set1
    DB2_DBX82_7 : BOOL ;	//Main contactor check-back signal
    DB2_DBX83_0 : BOOL ;	//Select function data set bit0
    DB2_DBX83_1 : BOOL ;	//Select function data set bit1
    DB2_DBX83_2 : BOOL ;	//Spare
    DB2_DBX83_3 : BOOL ;	//Spare
    DB2_DBX83_4 : BOOL ;	//Select fixed setpoint0
    DB2_DBX83_5 : BOOL ;	//Select fixed setpoint1
    DB2_DBX83_6 : BOOL ;	//Spare
    DB2_DBX83_7 : BOOL ;	//Spare
   END_STRUCT ;
   DB2_DBW84 : INT ;	//Motor speed reference
   DB2_DBW86 : INT ;
   DB2_DBW88 : INT ;
   DB2_DBW90 : INT ;
   DB2_DBW92 : INT ;
   DB2_DBW94 : INT ;
   DB2_DBW96 : INT ;
   DB2_DBW98 : INT ;
   DB2_DBW100 : INT ;
   DB2_DBW102 : INT ;
   DB2_DBW104 : INT ;
   DB2_DBW106 : INT ;
   DB2_DBW108 : INT ;
   DB2_DBW110 : INT ;
   DB2_DBW112 : INT ;
   DB2_DBW114 : INT ;
   DB2_DBW116 : INT ;
   DB2_DBW118 : INT ;
   CAGE_24_PREF_CONTROL_W1 : STRUCT
    DB2_DBX120_0 : BOOL ;	//Inching bit0
    DB2_DBX120_1 : BOOL ;	//Inching bit1
    DB2_DBX120_2 : BOOL ;	//Control requested
    DB2_DBX120_3 : BOOL ;	//Enable positive direction of rotation
    DB2_DBX120_4 : BOOL ;	//Enable negative direction of rotation
    DB2_DBX120_5 : BOOL ;	//Increase motorized potenziometer
    DB2_DBX120_6 : BOOL ;	//Decrease motorized potenziometer
    DB2_DBX120_7 : BOOL ;	//External fault1
    DB2_DBX121_0 : BOOL ;	//Off1
    DB2_DBX121_1 : BOOL ;	//Off2
    DB2_DBX121_2 : BOOL ;	//Off3
    DB2_DBX121_3 : BOOL ;	//Enable
    DB2_DBX121_4 : BOOL ;	//Enable ramp-function generetor
    DB2_DBX121_5 : BOOL ;	//Ramp-function generetor start
    DB2_DBX121_6 : BOOL ;	//Enable setpoint
    DB2_DBX121_7 : BOOL ;	//1Edge acknowledge
   END_STRUCT ;
   CAGE_24_PREF_CONTROL_W2 : STRUCT
    DB2_DBX122_0 : BOOL ;	//Enable speed controller droop
    DB2_DBX122_1 : BOOL ;	//Enable speed controller
    DB2_DBX122_2 : BOOL ;	//External fault2
    DB2_DBX122_3 : BOOL ;	//Master drive
    DB2_DBX122_4 : BOOL ;	//External alarm1
    DB2_DBX122_5 : BOOL ;	//External alarm2
    DB2_DBX122_6 : BOOL ;	//Select bico data set1
    DB2_DBX122_7 : BOOL ;	//Main contactor check-back signal
    DB2_DBX123_0 : BOOL ;	//Select function data set bit0
    DB2_DBX123_1 : BOOL ;	//Select function data set bit1
    DB2_DBX123_2 : BOOL ;	//Spare
    DB2_DBX123_3 : BOOL ;	//Spare
    DB2_DBX123_4 : BOOL ;	//Select fixed setpoint0
    DB2_DBX123_5 : BOOL ;	//Select fixed setpoint1
    DB2_DBX123_6 : BOOL ;	//Spare
    DB2_DBX123_7 : BOOL ;	//Spare
   END_STRUCT ;
   DB2_DBW124 : INT ;	//Motor speed reference
   DB2_DBW126 : INT ;
   DB2_DBW128 : INT ;
   DB2_DBW130 : INT ;
   DB2_DBW132 : INT ;
   DB2_DBW134 : INT ;
   DB2_DBW136 : INT ;
   DB2_DBW138 : INT ;
   DB2_DBW140 : INT ;
   DB2_DBW142 : INT ;
   DB2_DBW144 : INT ;
   DB2_DBW146 : INT ;
   DB2_DBW148 : INT ;
   DB2_DBW150 : INT ;
   DB2_DBW152 : INT ;
   DB2_DBW154 : INT ;
   DB2_DBW156 : INT ;
   DB2_DBW158 : INT ;
   CAGE_24_CONTROL_W1 : STRUCT
    DB2_DBX160_0 : BOOL ;	//Inching bit0
    DB2_DBX160_1 : BOOL ;	//Inching bit1
    DB2_DBX160_2 : BOOL ;	//Control requested
    DB2_DBX160_3 : BOOL ;	//Enable positive direction of rotation
    DB2_DBX160_4 : BOOL ;	//Enable negative direction of rotation
    DB2_DBX160_5 : BOOL ;	//Increase motorized potenziometer
    DB2_DBX160_6 : BOOL ;	//Decrease motorized potenziometer
    DB2_DBX160_7 : BOOL ;	//External fault1
    DB2_DBX161_0 : BOOL ;	//Off1
    DB2_DBX161_1 : BOOL ;	//Off2
    DB2_DBX161_2 : BOOL ;	//Off3
    DB2_DBX161_3 : BOOL ;	//Enable
    DB2_DBX161_4 : BOOL ;	//Enable ramp-function generetor
    DB2_DBX161_5 : BOOL ;	//Ramp-function generetor start
    DB2_DBX161_6 : BOOL ;	//Enable setpoint
    DB2_DBX161_7 : BOOL ;	//1Edge acknowledge
   END_STRUCT ;
   CAGE_24_CONTROL_W2 : STRUCT
    DB2_DBX162_0 : BOOL ;	//Enable speed controller droop
    DB2_DBX162_1 : BOOL ;	//Enable speed controller
    DB2_DBX162_2 : BOOL ;	//External fault2
    DB2_DBX162_3 : BOOL ;	//Master drive
    DB2_DBX162_4 : BOOL ;	//External alarm1
    DB2_DBX162_5 : BOOL ;	//External alarm2
    DB2_DBX162_6 : BOOL ;	//Select bico data set1
    DB2_DBX162_7 : BOOL ;	//Main contactor check-back signal
    DB2_DBX163_0 : BOOL ;	//Select function data set bit0
    DB2_DBX163_1 : BOOL ;	//Select function data set bit1
    DB2_DBX163_2 : BOOL ;	//Spare
    DB2_DBX163_3 : BOOL ;	//Spare
    DB2_DBX163_4 : BOOL ;	//Select fixed setpoint0
    DB2_DBX163_5 : BOOL ;	//Select fixed setpoint1
    DB2_DBX163_6 : BOOL ;	//Spare
    DB2_DBX163_7 : BOOL ;	//Spare
   END_STRUCT ;
   DB2_DBW164 : INT ;	//Motor speed reference
   DB2_DBW166 : INT ;
   DB2_DBW168 : INT ;
   DB2_DBW170 : INT ;
   DB2_DBW172 : INT ;
   DB2_DBW174 : INT ;
   DB2_DBW176 : INT ;
   DB2_DBW178 : INT ;
   DB2_DBW180 : INT ;
   DB2_DBW182 : INT ;
   DB2_DBW184 : INT ;
   DB2_DBW186 : INT ;
   DB2_DBW188 : INT ;
   DB2_DBW190 : INT ;
   DB2_DBW192 : INT ;
   DB2_DBW194 : INT ;
   DB2_DBW196 : INT ;
   DB2_DBW198 : INT ;
   CAGE_18_PREF_CONTROL_W1 : STRUCT
    DB2_DBX200_0 : BOOL ;	//Inching bit0
    DB2_DBX200_1 : BOOL ;	//Inching bit1
    DB2_DBX200_2 : BOOL ;	//Control requested
    DB2_DBX200_3 : BOOL ;	//Enable positive direction of rotation
    DB2_DBX200_4 : BOOL ;	//Enable negative direction of rotation
    DB2_DBX200_5 : BOOL ;	//Increase motorized potenziometer
    DB2_DBX200_6 : BOOL ;	//Decrease motorized potenziometer
    DB2_DBX200_7 : BOOL ;	//External fault1
    DB2_DBX201_0 : BOOL ;	//Off1
    DB2_DBX201_1 : BOOL ;	//Off2
    DB2_DBX201_2 : BOOL ;	//Off3
    DB2_DBX201_3 : BOOL ;	//Enable
    DB2_DBX201_4 : BOOL ;	//Enable ramp-function generetor
    DB2_DBX201_5 : BOOL ;	//Ramp-function generetor start
    DB2_DBX201_6 : BOOL ;	//Enable setpoint
    DB2_DBX201_7 : BOOL ;	//1Edge acknowledge
   END_STRUCT ;
   CAGE_18_PREF_CONTROL_W2 : STRUCT
    DB2_DBX202_0 : BOOL ;	//Enable speed controller droop
    DB2_DBX202_1 : BOOL ;	//Enable speed controller
    DB2_DBX202_2 : BOOL ;	//External fault2
    DB2_DBX202_3 : BOOL ;	//Master drive
    DB2_DBX202_4 : BOOL ;	//External alarm1
    DB2_DBX202_5 : BOOL ;	//External alarm2
    DB2_DBX202_6 : BOOL ;	//Select bico data set1
    DB2_DBX202_7 : BOOL ;	//Main contactor check-back signal
    DB2_DBX203_0 : BOOL ;	//Select function data set bit0
    DB2_DBX203_1 : BOOL ;	//Select function data set bit1
    DB2_DBX203_2 : BOOL ;	//Spare
    DB2_DBX203_3 : BOOL ;	//Spare
    DB2_DBX203_4 : BOOL ;	//Select fixed setpoint0
    DB2_DBX203_5 : BOOL ;	//Select fixed setpoint1
    DB2_DBX203_6 : BOOL ;	//Spare
    DB2_DBX203_7 : BOOL ;	//Spare
   END_STRUCT ;
   DB2_DBW204 : INT ;	//Motor speed reference
   DB2_DBW206 : INT ;
   DB2_DBW208 : INT ;
   DB2_DBW210 : INT ;
   DB2_DBW212 : INT ;
   DB2_DBW214 : INT ;
   DB2_DBW216 : INT ;
   DB2_DBW218 : INT ;
   DB2_DBW220 : INT ;
   DB2_DBW222 : INT ;
   DB2_DBW224 : INT ;
   DB2_DBW226 : INT ;
   DB2_DBW228 : INT ;
   DB2_DBW230 : INT ;
   DB2_DBW232 : INT ;
   DB2_DBW234 : INT ;
   DB2_DBW236 : INT ;
   DB2_DBW238 : INT ;
   CAGE_18_CONTROL_W1 : STRUCT
    DB2_DBX240_0 : BOOL ;	//Inching bit0
    DB2_DBX240_1 : BOOL ;	//Inching bit1
    DB2_DBX240_2 : BOOL ;	//Control requested
    DB2_DBX240_3 : BOOL ;	//Enable positive direction of rotation
    DB2_DBX240_4 : BOOL ;	//Enable negative direction of rotation
    DB2_DBX240_5 : BOOL ;	//Increase motorized potenziometer
    DB2_DBX240_6 : BOOL ;	//Decrease motorized potenziometer
    DB2_DBX240_7 : BOOL ;	//External fault1
    DB2_DBX241_0 : BOOL ;	//Off1
    DB2_DBX241_1 : BOOL ;	//Off2
    DB2_DBX241_2 : BOOL ;	//Off3
    DB2_DBX241_3 : BOOL ;	//Enable
    DB2_DBX241_4 : BOOL ;	//Enable ramp-function generetor
    DB2_DBX241_5 : BOOL ;	//Ramp-function generetor start
    DB2_DBX241_6 : BOOL ;	//Enable setpoint
    DB2_DBX241_7 : BOOL ;	//1Edge acknowledge
   END_STRUCT ;
   CAGE_18_CONTROL_W2 : STRUCT
    DB2_DBX242_0 : BOOL ;	//Enable speed controller droop
    DB2_DBX242_1 : BOOL ;	//Enable speed controller
    DB2_DBX242_2 : BOOL ;	//External fault2
    DB2_DBX242_3 : BOOL ;	//Master drive
    DB2_DBX242_4 : BOOL ;	//External alarm1
    DB2_DBX242_5 : BOOL ;	//External alarm2
    DB2_DBX242_6 : BOOL ;	//Select bico data set1
    DB2_DBX242_7 : BOOL ;	//Main contactor check-back signal
    DB2_DBX243_0 : BOOL ;	//Select function data set bit0
    DB2_DBX243_1 : BOOL ;	//Select function data set bit1
    DB2_DBX243_2 : BOOL ;	//Spare
    DB2_DBX243_3 : BOOL ;	//Spare
    DB2_DBX243_4 : BOOL ;	//Select fixed setpoint0
    DB2_DBX243_5 : BOOL ;	//Select fixed setpoint1
    DB2_DBX243_6 : BOOL ;	//Spare
    DB2_DBX243_7 : BOOL ;	//Spare
   END_STRUCT ;
   DB2_DBW244 : INT ;	//Motor speed reference
   DB2_DBW246 : INT ;
   DB2_DBW248 : INT ;
   DB2_DBW250 : INT ;
   DB2_DBW252 : INT ;
   DB2_DBW254 : INT ;
   DB2_DBW256 : INT ;
   DB2_DBW258 : INT ;
   DB2_DBW260 : INT ;
   DB2_DBW262 : INT ;
   DB2_DBW264 : INT ;
   DB2_DBW266 : INT ;
   DB2_DBW268 : INT ;
   DB2_DBW270 : INT ;
   DB2_DBW272 : INT ;
   DB2_DBW274 : INT ;
   DB2_DBW276 : INT ;
   DB2_DBW278 : INT ;
   CAGE_12_PREF_CONTROL_W1 : STRUCT
    DB2_DBX280_0 : BOOL ;	//Inching bit0
    DB2_DBX280_1 : BOOL ;	//Inching bit1
    DB2_DBX280_2 : BOOL ;	//Control requested
    DB2_DBX280_3 : BOOL ;	//Enable positive direction of rotation
    DB2_DBX280_4 : BOOL ;	//Enable negative direction of rotation
    DB2_DBX280_5 : BOOL ;	//Increase motorized potenziometer
    DB2_DBX280_6 : BOOL ;	//Decrease motorized potenziometer
    DB2_DBX280_7 : BOOL ;	//External fault1
    DB2_DBX281_0 : BOOL ;	//Off1
    DB2_DBX281_1 : BOOL ;	//Off2
    DB2_DBX281_2 : BOOL ;	//Off3
    DB2_DBX281_3 : BOOL ;	//Enable
    DB2_DBX281_4 : BOOL ;	//Enable ramp-function generetor
    DB2_DBX281_5 : BOOL ;	//Ramp-function generetor start
    DB2_DBX281_6 : BOOL ;	//Enable setpoint
    DB2_DBX281_7 : BOOL ;	//1Edge acknowledge
   END_STRUCT ;
   CAGE_12_PREF_CONTROL_W2 : STRUCT
    DB2_DBX282_0 : BOOL ;	//Enable speed controller droop
    DB2_DBX282_1 : BOOL ;	//Enable speed controller
    DB2_DBX282_2 : BOOL ;	//External fault2
    DB2_DBX282_3 : BOOL ;	//Master drive
    DB2_DBX282_4 : BOOL ;	//External alarm1
    DB2_DBX282_5 : BOOL ;	//External alarm2
    DB2_DBX282_6 : BOOL ;	//Select bico data set1
    DB2_DBX282_7 : BOOL ;	//Main contactor check-back signal
    DB2_DBX283_0 : BOOL ;	//Select function data set bit0
    DB2_DBX283_1 : BOOL ;	//Select function data set bit1
    DB2_DBX283_2 : BOOL ;	//Spare
    DB2_DBX283_3 : BOOL ;	//Spare
    DB2_DBX283_4 : BOOL ;	//Select fixed setpoint0
    DB2_DBX283_5 : BOOL ;	//Select fixed setpoint1
    DB2_DBX283_6 : BOOL ;	//Spare
    DB2_DBX283_7 : BOOL ;	//Spare
   END_STRUCT ;
   DB2_DBW284 : INT ;	//Motor speed reference
   DB2_DBW286 : INT ;
   DB2_DBW288 : INT ;
   DB2_DBW290 : INT ;
   DB2_DBW292 : INT ;
   DB2_DBW294 : INT ;
   DB2_DBW296 : INT ;
   DB2_DBW298 : INT ;
   DB2_DBW300 : INT ;
   DB2_DBW302 : INT ;
   DB2_DBW304 : INT ;
   DB2_DBW306 : INT ;
   DB2_DBW308 : INT ;
   DB2_DBW310 : INT ;
   DB2_DBW312 : INT ;
   DB2_DBW314 : INT ;
   DB2_DBW316 : INT ;
   DB2_DBW318 : INT ;
   CAGE_12_CONTROL_W1 : STRUCT
    DB2_DBX320_0 : BOOL ;	//Inching bit0
    DB2_DBX320_1 : BOOL ;	//Inching bit1
    DB2_DBX320_2 : BOOL ;	//Control requested
    DB2_DBX320_3 : BOOL ;	//Enable positive direction of rotation
    DB2_DBX320_4 : BOOL ;	//Enable negative direction of rotation
    DB2_DBX320_5 : BOOL ;	//Increase motorized potenziometer
    DB2_DBX320_6 : BOOL ;	//Decrease motorized potenziometer
    DB2_DBX320_7 : BOOL ;	//External fault1
    DB2_DBX321_0 : BOOL ;	//Off1
    DB2_DBX321_1 : BOOL ;	//Off2
    DB2_DBX321_2 : BOOL ;	//Off3
    DB2_DBX321_3 : BOOL ;	//Enable
    DB2_DBX321_4 : BOOL ;	//Enable ramp-function generetor
    DB2_DBX321_5 : BOOL ;	//Ramp-function generetor start
    DB2_DBX321_6 : BOOL ;	//Enable setpoint
    DB2_DBX321_7 : BOOL ;	//1Edge acknowledge
   END_STRUCT ;
   CAGE_12_CONTROL_W2 : STRUCT
    DB2_DBX322_0 : BOOL ;	//Enable speed controller droop
    DB2_DBX322_1 : BOOL ;	//Enable speed controller
    DB2_DBX322_2 : BOOL ;	//External fault2
    DB2_DBX322_3 : BOOL ;	//Master drive
    DB2_DBX322_4 : BOOL ;	//External alarm1
    DB2_DBX322_5 : BOOL ;	//External alarm2
    DB2_DBX322_6 : BOOL ;	//Select bico data set1
    DB2_DBX322_7 : BOOL ;	//Main contactor check-back signal
    DB2_DBX323_0 : BOOL ;	//Select function data set bit0
    DB2_DBX323_1 : BOOL ;	//Select function data set bit1
    DB2_DBX323_2 : BOOL ;	//Spare
    DB2_DBX323_3 : BOOL ;	//Spare
    DB2_DBX323_4 : BOOL ;	//Select fixed setpoint0
    DB2_DBX323_5 : BOOL ;	//Select fixed setpoint1
    DB2_DBX323_6 : BOOL ;	//Spare
    DB2_DBX323_7 : BOOL ;	//Spare
   END_STRUCT ;
   DB2_DBW324 : INT ;	//Motor speed reference
   DB2_DBW326 : INT ;
   DB2_DBW328 : INT ;
   DB2_DBW330 : INT ;
   DB2_DBW332 : INT ;
   DB2_DBW334 : INT ;
   DB2_DBW336 : INT ;
   DB2_DBW338 : INT ;
   DB2_DBW340 : INT ;
   DB2_DBW342 : INT ;
   DB2_DBW344 : INT ;
   DB2_DBW346 : INT ;
   DB2_DBW348 : INT ;
   DB2_DBW350 : INT ;
   DB2_DBW352 : INT ;
   DB2_DBW354 : INT ;
   DB2_DBW356 : INT ;
   DB2_DBW358 : INT ;
   CAGE_6_CONTROL_W1 : STRUCT
    DB2_DBX360_0 : BOOL ;	//Inching bit0
    DB2_DBX360_1 : BOOL ;	//Inching bit1
    DB2_DBX360_2 : BOOL ;	//Control requested
    DB2_DBX360_3 : BOOL ;	//Enable positive direction of rotation
    DB2_DBX360_4 : BOOL ;	//Enable negative direction of rotation
    DB2_DBX360_5 : BOOL ;	//Increase motorized potenziometer
    DB2_DBX360_6 : BOOL ;	//Decrease motorized potenziometer
    DB2_DBX360_7 : BOOL ;	//External fault1
    DB2_DBX361_0 : BOOL ;	//Off1
    DB2_DBX361_1 : BOOL ;	//Off2
    DB2_DBX361_2 : BOOL ;	//Off3
    DB2_DBX361_3 : BOOL ;	//Enable
    DB2_DBX361_4 : BOOL ;	//Enable ramp-function generetor
    DB2_DBX361_5 : BOOL ;	//Ramp-function generetor start
    DB2_DBX361_6 : BOOL ;	//Enable setpoint
    DB2_DBX361_7 : BOOL ;	//1Edge acknowledge
   END_STRUCT ;
   CAGE_6_CONTROL_W2 : STRUCT
    DB2_DBX362_0 : BOOL ;	//Enable speed controller droop
    DB2_DBX362_1 : BOOL ;	//Enable speed controller
    DB2_DBX362_2 : BOOL ;	//External fault2
    DB2_DBX362_3 : BOOL ;	//Master drive
    DB2_DBX362_4 : BOOL ;	//External alarm1
    DB2_DBX362_5 : BOOL ;	//External alarm2
    DB2_DBX362_6 : BOOL ;	//Select bico data set1
    DB2_DBX362_7 : BOOL ;	//Main contactor check-back signal
    DB2_DBX363_0 : BOOL ;	//Select function data set bit0
    DB2_DBX363_1 : BOOL ;	//Select function data set bit1
    DB2_DBX363_2 : BOOL ;	//Spare
    DB2_DBX363_3 : BOOL ;	//Spare
    DB2_DBX363_4 : BOOL ;	//Select fixed setpoint0
    DB2_DBX363_5 : BOOL ;	//Select fixed setpoint1
    DB2_DBX363_6 : BOOL ;	//Spare
    DB2_DBX363_7 : BOOL ;	//Spare
   END_STRUCT ;
   DB2_DBW364 : INT ;	//Motor speed reference
   DB2_DBW366 : INT ;
   DB2_DBW368 : INT ;
   DB2_DBW370 : INT ;
   DB2_DBW372 : INT ;
   DB2_DBW374 : INT ;
   DB2_DBW376 : INT ;
   DB2_DBW378 : INT ;
   DB2_DBW380 : INT ;
   DB2_DBW382 : INT ;
   DB2_DBW384 : INT ;
   DB2_DBW386 : INT ;
   DB2_DBW388 : INT ;
   DB2_DBW390 : INT ;
   DB2_DBW392 : INT ;
   DB2_DBW394 : INT ;
   DB2_DBW396 : INT ;
   DB2_DBW398 : INT ;
   SPARE_CONTROL_W1 : STRUCT
    DB2_DBX400_0 : BOOL ;	//Inching bit0
    DB2_DBX400_1 : BOOL ;	//Inching bit1
    DB2_DBX400_2 : BOOL ;	//Control requested
    DB2_DBX400_3 : BOOL ;	//Enable positive direction of rotation
    DB2_DBX400_4 : BOOL ;	//Enable negative direction of rotation
    DB2_DBX400_5 : BOOL ;	//Increase motorized potenziometer
    DB2_DBX400_6 : BOOL ;	//Decrease motorized potenziometer
    DB2_DBX400_7 : BOOL ;	//External fault1
    DB2_DBX401_0 : BOOL ;	//Off1
    DB2_DBX401_1 : BOOL ;	//Off2
    DB2_DBX401_2 : BOOL ;	//Off3
    DB2_DBX401_3 : BOOL ;	//Enable
    DB2_DBX401_4 : BOOL ;	//Enable ramp-function generetor
    DB2_DBX401_5 : BOOL ;	//Ramp-function generetor start
    DB2_DBX401_6 : BOOL ;	//Enable setpoint
    DB2_DBX401_7 : BOOL ;	//1Edge acknowledge
   END_STRUCT ;
   SPARE_CONTROL_W2 : STRUCT
    DB2_DBX402_0 : BOOL ;	//Enable speed controller droop
    DB2_DBX402_1 : BOOL ;	//Enable speed controller
    DB2_DBX402_2 : BOOL ;	//External fault2
    DB2_DBX402_3 : BOOL ;	//Master drive
    DB2_DBX402_4 : BOOL ;	//External alarm1
    DB2_DBX402_5 : BOOL ;	//External alarm2
    DB2_DBX402_6 : BOOL ;	//Select bico data set1
    DB2_DBX402_7 : BOOL ;	//Main contactor check-back signal
    DB2_DBX403_0 : BOOL ;	//Select function data set bit0
    DB2_DBX403_1 : BOOL ;	//Select function data set bit1
    DB2_DBX403_2 : BOOL ;	//Spare
    DB2_DBX403_3 : BOOL ;	//Spare
    DB2_DBX403_4 : BOOL ;	//Select fixed setpoint0
    DB2_DBX403_5 : BOOL ;	//Select fixed setpoint1
    DB2_DBX403_6 : BOOL ;	//Spare
    DB2_DBX403_7 : BOOL ;	//Spare
   END_STRUCT ;
   DB2_DBW404 : INT ;
   DB2_DBW406 : INT ;
   DB2_DBW408 : INT ;
   DB2_DBW410 : INT ;
   DB2_DBW412 : INT ;
   DB2_DBW414 : INT ;
   DB2_DBW416 : INT ;
   DB2_DBW418 : INT ;
   DB2_DBW420 : INT ;
   DB2_DBW422 : INT ;
   DB2_DBW424 : INT ;
   DB2_DBW426 : INT ;
   DB2_DBW428 : INT ;
   DB2_DBW430 : INT ;
   DB2_DBW432 : INT ;
   DB2_DBW434 : INT ;
   DB2_DBW436 : INT ;
   DB2_DBW438 : INT ;
   DB2_DBW440 : INT ;
   DB2_DBW442 : INT ;
   DB2_DBW444 : INT ;
   DB2_DBW446 : INT ;
   DB2_DBW448 : INT ;
   DB2_DBW450 : INT ;
   DB2_DBW452 : INT ;
   DB2_DBW454 : INT ;
   DB2_DBW456 : INT ;
   DB2_DBW458 : INT ;
   DB2_DBW460 : INT ;
   DB2_DBW462 : INT ;
   DB2_DBW464 : INT ;
   DB2_DBW466 : INT ;
   DB2_DBW468 : INT ;
   DB2_DBW470 : INT ;
   DB2_DBW472 : INT ;
   DB2_DBW474 : INT ;
   DB2_DBW476 : INT ;
   DB2_DBW478 : INT ;
   DB2_DBW480 : INT ;
   DB2_DBW482 : INT ;
   DB2_DBW484 : INT ;
   DB2_DBW486 : INT ;
   DB2_DBW488 : INT ;
   DB2_DBW490 : INT ;
   DB2_DBW492 : INT ;
   DB2_DBW494 : INT ;
   DB2_DBW496 : INT ;
   DB2_DBW498 : INT ;
   PKW_WRITE_CAGE24 : STRUCT
    DB2_DBW500 : INT ;	//PKE
    DB2_DBW502 : INT ;	//IND
    DB2_DBW504 : INT ;	//PWE1
    DB2_DBW506 : INT ;	//PWE2
   END_STRUCT ;
   DB2_DBW508 : INT ;	//Spare
   PKW_WRITE_CAGE18 : STRUCT
    DB2_DBW510 : INT ;	//PKE
    DB2_DBW512 : INT ;	//IND
    DB2_DBW514 : INT ;	//PWE1
    DB2_DBW516 : INT ;	//PWE2
   END_STRUCT ;
   DB2_DBW518 : INT ;	//Spare
   PKW_WRITE_CAGE12 : STRUCT
    DB2_DBW520 : INT ;	//PKE
    DB2_DBW522 : INT ;	//IND
    DB2_DBW524 : INT ;	//PWE1
    DB2_DBW526 : INT ;	//PWE2
   END_STRUCT ;
   DB2_DBW528 : INT ;	//Spare
   PKW_WRITE_CAGE6 : STRUCT
    DB2_DBW530 : INT ;	//PKE
    DB2_DBW532 : INT ;	//IND
    DB2_DBW534 : INT ;	//PWE1
    DB2_DBW536 : INT ;	//PWE2
   END_STRUCT ;
   DB2_DBW538 : INT ;	//Spare
  END_STRUCT ;	
BEGIN
   TRAVERSE_CONTROL_W1.DB2_DBX0_2 := TRUE;
   TRAVERSE_CONTROL_W1.DB2_DBX1_2 := TRUE;
   DB2_DBW6 := 605;
   BOBBIN_CONTROL_W1.DB2_DBX40_2 := TRUE;
   BOBBIN_CONTROL_W1.DB2_DBX41_0 := TRUE;
   BOBBIN_CONTROL_W1.DB2_DBX41_2 := TRUE;
   BOBBIN_CONTROL_W1.DB2_DBX41_3 := TRUE;
   DB2_DBW44 := 1638;
   DB2_DBW46 := 2092;
   CAPSTAN_CONTROL_W1.DB2_DBX80_2 := TRUE;
   CAPSTAN_CONTROL_W1.DB2_DBX81_2 := TRUE;
   CAGE_24_PREF_CONTROL_W1.DB2_DBX120_2 := TRUE;
   CAGE_24_PREF_CONTROL_W1.DB2_DBX121_2 := TRUE;
   CAGE_24_CONTROL_W1.DB2_DBX160_2 := TRUE;
   CAGE_24_CONTROL_W1.DB2_DBX161_2 := TRUE;
   CAGE_18_PREF_CONTROL_W1.DB2_DBX200_2 := TRUE;
   CAGE_18_PREF_CONTROL_W1.DB2_DBX201_2 := TRUE;
   CAGE_18_CONTROL_W1.DB2_DBX240_2 := TRUE;
   CAGE_18_CONTROL_W1.DB2_DBX241_2 := TRUE;
   CAGE_12_PREF_CONTROL_W1.DB2_DBX280_2 := TRUE;
   CAGE_12_PREF_CONTROL_W1.DB2_DBX281_2 := TRUE;
   CAGE_12_CONTROL_W1.DB2_DBX320_2 := TRUE;
   CAGE_12_CONTROL_W1.DB2_DBX321_2 := TRUE;
   CAGE_6_CONTROL_W1.DB2_DBX360_2 := TRUE;
   CAGE_6_CONTROL_W1.DB2_DBX361_2 := TRUE;
   SPARE_CONTROL_W1.DB2_DBX400_2 := TRUE;
   SPARE_CONTROL_W1.DB2_DBX401_2 := TRUE;
   DB2_DBW406 := 65;
   DB2_DBW410 := 8710;
   DB2_DBW416 := 65;
   DB2_DBW420 := 8710;
   DB2_DBW426 := 65;
   DB2_DBW430 := 8710;
   DB2_DBW436 := 65;
   PKW_WRITE_CAGE24.DB2_DBW500 := 8709;
   PKW_WRITE_CAGE18.DB2_DBW510 := 8709;
   PKW_WRITE_CAGE12.DB2_DBW520 := 8709;
   PKW_WRITE_CAGE12.DB2_DBW526 := 1;
   PKW_WRITE_CAGE6.DB2_DBW530 := 8709;
END_DATA_BLOCK

DATA_BLOCK "Profibus SFC Alarm"	// DB 3
TITLE = PROFIBUS SFC ALARM DATA BLOCK
AUTHOR : Milesi
VERSION : 0.1
  STRUCT
   DB3_DBW0 : INT ;	//PZD_Return value reading take-up traverse address 3
   DB3_DBW2 : INT ;	//PZD_Return value writing take-up traverse address 3
   DB3_DBW4 : INT ;	//PZD_Return value reading take-up bobbin motor address 4
   DB3_DBW6 : INT ;	//PZD_Return value writing take-up bobbin motor address 4
   DB3_DBW8 : INT ;	//PZD_Return value reading capstan motor address 5
   DB3_DBW10 : INT ;	//PZD_Return value writing capstan motor address 5
   DB3_DBW12 : INT ;	//PZD_Return value reading cage 18 preforming motor address 8
   DB3_DBW14 : INT ;	//PZD_Return value writing cage 18 preforming motor address 8
   DB3_DBW16 : INT ;	//PZD_Return value reading cage 18 motor address 9
   DB3_DBW18 : INT ;	//PZD_Return value writing cage 18 motor address 9
   DB3_DBW20 : INT ;	//PZD_Return value reading cage 12 preforming motor address 10
   DB3_DBW22 : INT ;	//PZD_Return value writing cage 12 preforming motor address 10
   DB3_DBW24 : INT ;	//PZD_Return value reading cage 12 motor address 11
   DB3_DBW26 : INT ;	//PZD_Return value writing cage 12 motor address 11
   DB3_DBW28 : INT ;	//PZD_Return value reading cage 6 motor address 12
   DB3_DBW30 : INT ;	//PZD_Return value writing cage 6 motor address 12
   DB3_DBW32 : INT ;	//PZD_Return value reading cage 24 preforming motor address 6
   DB3_DBW34 : INT ;	//PZD_Return value writing cage 24 preforming motor address 6
   DB3_DBW36 : INT ;	//PZD_Return value reading cage 24 motor address 7
   DB3_DBW38 : INT ;	//PZD_Return value writing cage 24 motor address 7
   DB3_DBW40 : INT ;	//PZD_Return value reading pay-off traverse address 3
   DB3_DBW42 : INT ;	//PZD_Return value writing pay-off traverse address 3
   DB3_DBW44 : INT ;
   DB3_DBW46 : INT ;
   DB3_DBW48 : INT ;	//PKW_Return value reading cage 24 motor address 7
   DB3_DBW50 : INT ;	//PKW_Return value writing cage 24 motor address 7
   DB3_DBW52 : INT ;	//PKW_Return value reading cage 18 motor address 9
   DB3_DBW54 : INT ;	//PKW_Return value writing cage 18 motor address 9
   DB3_DBW56 : INT ;	//PKW_Return value reading cage 12 motor address 11
   DB3_DBW58 : INT ;	//PKW_Return value writing cage 12 motor address 11
   DB3_DBW60 : INT ;	//PKW_Return value reading cage 6 motor address 12
   DB3_DBW62 : INT ;	//PKW_Return value writing cage 6 motor address 12
  END_STRUCT ;	
BEGIN
   DB3_DBW24 := -32624;
END_DATA_BLOCK

DATA_BLOCK "Take-up traverse"	// DB 5
TITLE = TAKE-UP TRAVERSE DATA BLOCK
AUTHOR : Milesi
VERSION : 0.1
  STRUCT
   HMI_Bit : STRUCT
    DB5_DBX0_0 : BOOL ;
    DB5_DBX0_1 : BOOL ;
    DB5_DBX0_2 : BOOL ;	//Home positioning on to HMI
    DB5_DBX0_3 : BOOL ;
    DB5_DBX0_4 : BOOL ;
    DB5_DBX0_5 : BOOL ;
    DB5_DBX0_6 : BOOL ;
    DB5_DBX0_7 : BOOL ;
    DB5_DBX1_0 : BOOL ;	//Right direction impulse from HMI
    DB5_DBX1_1 : BOOL ;	//Left direction impulse from HMI
    DB5_DBX1_2 : BOOL ;	//Home positioning impulse from HMI
    DB5_DBX1_3 : BOOL ;
    DB5_DBX1_4 : BOOL ;
    DB5_DBX1_5 : BOOL ;
    DB5_DBX1_6 : BOOL ;
    DB5_DBX1_7 : BOOL ;
   END_STRUCT ;
   DB5_DBW2 : INT ;
   DB5_DBW4 : INT ;
   DB5_DBW6 : INT ;
   DB5_DBW8 : INT ;
   DB5_DBW10 : INT ;
   DB5_DBW12 : INT ;
   DB5_DBW14 : INT ;
   DB5_DBW16 : INT ;
   DB5_DBW18 : INT ;
   DB5_DBD20 : REAL ;	//Lay set from HMI
   DB5_DBD24 : REAL ;	//Left flange limit set from HMI
   DB5_DBD28 : REAL ;	//Right flange limit set from HMI
   DB5_DBD32 : REAL ;	//Encoder position mm to HMI
   DB5_DBD36 : REAL ;	//Speed reference
   DB5_DBD40 : REAL ;	//Encoder position
   DB5_DBD44 : DINT ;	//Encoder counter hold
   DB5_DBD48 : REAL ;	//Inversion delay count set from HMI
   DB5_DBD52 : REAL ;	//Inversion delay count read to HMI
   DB5_DBD56 : REAL ;
   DB5_DBD60 : REAL ;
   DB5_DBD64 : REAL ;
   DB5_DBD68 : REAL ;
   DB5_DBD72 : REAL ;
   DB5_DBD76 : REAL ;
   DB5_DBD80 : REAL ;
   DB5_DBD84 : REAL ;
   DB5_DBD88 : REAL ;
   DB5_DBD92 : REAL ;
   DB5_DBD96 : REAL ;
   DB5_DBD100 : REAL ;
   DB5_DBD104 : REAL ;
   DB5_DBD108 : REAL ;
   DB5_DBD112 : REAL ;
   DB5_DBD116 : REAL ;
   DB5_DBD120 : REAL ;
   DB5_DBD124 : REAL ;
   DB5_DBD128 : REAL ;
   DB5_DBD132 : REAL ;
   DB5_DBD136 : REAL ;
   DB5_DBD140 : REAL ;
   DB5_DBD144 : REAL ;
   DB5_DBD148 : REAL ;
   DB5_DBD152 : REAL ;
   DB5_DBD156 : REAL ;
   DB5_DBD160 : REAL ;
   DB5_DBD164 : REAL ;
   DB5_DBD168 : REAL ;
   DB5_DBD172 : REAL ;
   DB5_DBD176 : REAL ;
   DB5_DBD180 : REAL ;
   DB5_DBD184 : REAL ;
   DB5_DBD188 : REAL ;	//Motor rpm to HMI
   DB5_DBD192 : REAL ;	//Motor current to HMI
   DB5_DBD196 : REAL ;	//Motor voltage to HMI
   DB5_DBD200 : REAL ;	//Speed reference to drive
   DB5_DBD204 : REAL ;
   DB5_DBD208 : REAL ;
   DB5_DBD212 : REAL ;
   DB5_DBD216 : REAL ;
   DB5_DBD220 : REAL ;
   DB5_DBD224 : REAL ;
   DB5_DBD228 : REAL ;
   DB5_DBD232 : REAL ;
   DB5_DBD236 : REAL ;
   DB5_DBD240 : REAL ;
   DB5_DBD244 : REAL ;
   DB5_DBD248 : REAL ;
   DB5_DBD252 : REAL ;
   DB5_DBD256 : REAL ;
   DB5_DBD260 : REAL ;
   DB5_DBD264 : REAL ;
   DB5_DBD268 : REAL ;
   DB5_DBD272 : REAL ;
   DB5_DBD276 : REAL ;
  END_STRUCT ;	
BEGIN
   HMI_Bit.DB5_DBX0_1 := TRUE;
   DB5_DBD20 := 3.000000e+01;
   DB5_DBD24 := 5.300000e+02;
   DB5_DBD28 := -2.400000e+02;
   DB5_DBD44 := L#-67180;
END_DATA_BLOCK

DATA_BLOCK "Take-up"	// DB 7
TITLE = TAKE-UP DATA BLOCK
AUTHOR : Milesi
VERSION : 0.1
  STRUCT
   HMI_Bit : STRUCT
    DB7_DBX0_0 : BOOL ;
    DB7_DBX0_1 : BOOL ;
    DB7_DBX0_2 : BOOL ;
    DB7_DBX0_3 : BOOL ;
    DB7_DBX0_4 : BOOL ;
    DB7_DBX0_5 : BOOL ;
    DB7_DBX0_6 : BOOL ;
    DB7_DBX0_7 : BOOL ;
    DB7_DBX1_0 : BOOL ;
    DB7_DBX1_1 : BOOL ;
    DB7_DBX1_2 : BOOL ;
    DB7_DBX1_3 : BOOL ;
    DB7_DBX1_4 : BOOL ;
    DB7_DBX1_5 : BOOL ;
    DB7_DBX1_6 : BOOL ;
    DB7_DBX1_7 : BOOL ;
   END_STRUCT ;
   DB7_DBW2 : INT ;
   DB7_DBW4 : INT ;
   DB7_DBW6 : INT ;
   DB7_DBW8 : INT ;
   DB7_DBW10 : INT ;
   DB7_DBW12 : INT ;
   DB7_DBW14 : INT ;
   DB7_DBW16 : INT ;
   DB7_DBW18 : INT ;
   DB7_DBD20 : REAL ;	//Pull set from HMI
   DB7_DBD24 : REAL ;	//Stall pull set from HMI
   DB7_DBD28 : REAL ;	//Flange diameter set from HMI
   DB7_DBD32 : REAL ;	//Static friction set from HMI
   DB7_DBD36 : REAL ;	//Dynamic friction set from HMI
   DB7_DBD40 : REAL ;	//Rpm to HMI
   DB7_DBD44 : REAL ;
   DB7_DBD48 : REAL ;	//Jog rpm from HMI
   DB7_DBD52 : REAL ;	//Flange diameter / 2 to HMI
   DB7_DBD56 : REAL ;	//Real diameter
   DB7_DBD60 : REAL ;	//Diameter filter aux 1
   DB7_DBD64 : REAL ;	//Diameter filter aux 2
   DB7_DBD68 : REAL ;	//Pull reference
   DB7_DBD72 : REAL ;	//Static compensation
   DB7_DBD76 : REAL ;	//Dynamic compensation
   DB7_DBD80 : REAL ;
   DB7_DBD84 : REAL ;	//K pull adjustment
   DB7_DBD88 : REAL ;
   DB7_DBD92 : REAL ;
   DB7_DBD96 : REAL ;
   DB7_DBD100 : REAL ;
   DB7_DBD104 : REAL ;
   DB7_DBD108 : REAL ;
   DB7_DBD112 : REAL ;
   DB7_DBD116 : REAL ;
   DB7_DBD120 : REAL ;
   DB7_DBD124 : REAL ;
   DB7_DBD128 : REAL ;
   DB7_DBD132 : REAL ;
   DB7_DBD136 : REAL ;
   DB7_DBD140 : REAL ;
   DB7_DBD144 : REAL ;
   DB7_DBD148 : REAL ;
   DB7_DBD152 : REAL ;
   DB7_DBD156 : REAL ;
   DB7_DBD160 : REAL ;
   DB7_DBD164 : REAL ;
   DB7_DBD168 : REAL ;
   DB7_DBD172 : REAL ;
   DB7_DBD176 : REAL ;
   DB7_DBD180 : REAL ;
   DB7_DBD184 : REAL ;
   DB7_DBD188 : REAL ;	//Motor rpm to HMI
   DB7_DBD192 : REAL ;	//Motor current to HMI
   DB7_DBD196 : REAL ;	//Motor voltage to HMI
   DB7_DBD200 : REAL ;	//Speed reference to drive
   DB7_DBD204 : REAL ;
   DB7_DBD208 : REAL ;	//Pull reference to drive
   DB7_DBD212 : REAL ;
   DB7_DBD216 : REAL ;
   DB7_DBD220 : REAL ;
   DB7_DBD224 : REAL ;
   DB7_DBD228 : REAL ;
   DB7_DBD232 : REAL ;
   DB7_DBD236 : REAL ;
   DB7_DBD240 : REAL ;
   DB7_DBD244 : REAL ;
   DB7_DBD248 : REAL ;
   DB7_DBD252 : REAL ;
   DB7_DBD256 : REAL ;
   DB7_DBD260 : REAL ;
   DB7_DBD264 : REAL ;
   DB7_DBD268 : REAL ;
   DB7_DBD272 : REAL ;
   DB7_DBD276 : REAL ;
  END_STRUCT ;	
BEGIN
   DB7_DBW2 := 3;
   DB7_DBD20 := 6.500000e+01;
   DB7_DBD24 := 4.000000e+01;
   DB7_DBD28 := 1.600000e+03;
   DB7_DBD44 := 2.240000e+02;
   DB7_DBD48 := 3.000000e+00;
   DB7_DBD52 := 8.000000e+02;
   DB7_DBD56 := 1.100311e+03;
   DB7_DBD68 := 2.092478e+03;
   DB7_DBD80 := 1.000000e+01;
   DB7_DBD84 := 1.400000e+00;
   DB7_DBD88 := 6.203613e+00;
   DB7_DBD92 := 5.065430e+00;
   DB7_DBD96 := 2.010498e+00;
   DB7_DBD100 := 1.913033e+01;
   DB7_DBD192 := 2.739990e+00;
   DB7_DBD196 := 1.279297e+01;
END_DATA_BLOCK

DATA_BLOCK "Capstan"	// DB 9
TITLE = CAPSTAN DATA BLOCK
AUTHOR : Milesi
VERSION : 0.1
  STRUCT
   HMI_Bit : STRUCT
    DB9_DBX0_0 : BOOL ;
    DB9_DBX0_1 : BOOL ;
    DB9_DBX0_2 : BOOL ;
    DB9_DBX0_3 : BOOL ;
    DB9_DBX0_4 : BOOL ;
    DB9_DBX0_5 : BOOL ;
    DB9_DBX0_6 : BOOL ;
    DB9_DBX0_7 : BOOL ;
    DB9_DBX1_0 : BOOL ;
    DB9_DBX1_1 : BOOL ;
    DB9_DBX1_2 : BOOL ;
    DB9_DBX1_3 : BOOL ;
    DB9_DBX1_4 : BOOL ;
    DB9_DBX1_5 : BOOL ;
    DB9_DBX1_6 : BOOL ;
    DB9_DBX1_7 : BOOL ;
   END_STRUCT ;
   DB9_DBW2 : INT ;
   DB9_DBW4 : INT ;
   DB9_DBW6 : INT ;
   DB9_DBW8 : INT ;
   DB9_DBW10 : INT ;
   DB9_DBW12 : INT ;
   DB9_DBW14 : INT ;
   DB9_DBW16 : INT ;
   DB9_DBW18 : INT ;
   DB9_DBD20 : REAL ;	//Jog speed from HMI
   DB9_DBD24 : REAL ;
   DB9_DBD28 : REAL ;
   DB9_DBD32 : REAL ;
   DB9_DBD36 : REAL ;
   DB9_DBD40 : REAL ;
   DB9_DBD44 : REAL ;
   DB9_DBD48 : REAL ;
   DB9_DBD52 : REAL ;
   DB9_DBD56 : REAL ;
   DB9_DBD60 : REAL ;	//Added value
   DB9_DBD64 : REAL ;	//Counter increase
   DB9_DBD68 : REAL ;	//Capstan actual speed
   DB9_DBD72 : REAL ;	//Normal stop brake constant from HMI
   DB9_DBD76 : REAL ;	//Emergency stop brake constant from HMI
   DB9_DBD80 : REAL ;	//Missing power supply stop brake constant from HMI
   DB9_DBD84 : REAL ;
   DB9_DBD88 : REAL ;
   DB9_DBD92 : REAL ;
   DB9_DBD96 : REAL ;
   DB9_DBD100 : REAL ;
   DB9_DBD104 : REAL ;
   DB9_DBD108 : REAL ;
   DB9_DBD112 : REAL ;
   DB9_DBD116 : REAL ;
   DB9_DBD120 : REAL ;
   DB9_DBD124 : REAL ;
   DB9_DBD128 : REAL ;
   DB9_DBD132 : REAL ;
   DB9_DBD136 : REAL ;
   DB9_DBD140 : REAL ;
   DB9_DBD144 : REAL ;
   DB9_DBD148 : REAL ;
   DB9_DBD152 : REAL ;
   DB9_DBD156 : REAL ;
   DB9_DBD160 : REAL ;
   DB9_DBD164 : REAL ;
   DB9_DBD168 : REAL ;
   DB9_DBD172 : REAL ;
   DB9_DBD176 : REAL ;
   DB9_DBD180 : REAL ;
   DB9_DBD184 : REAL ;
   DB9_DBD188 : REAL ;	//Motor rpm to HMI
   DB9_DBD192 : REAL ;	//Motor current to HMI
   DB9_DBD196 : REAL ;	//Motor voltage to HMI
   DB9_DBD200 : REAL ;	//Speed reference to drive
   DB9_DBD204 : REAL ;
   DB9_DBD208 : REAL ;
   DB9_DBD212 : REAL ;
   DB9_DBD216 : REAL ;
   DB9_DBD220 : REAL ;
   DB9_DBD224 : REAL ;
   DB9_DBD228 : REAL ;
   DB9_DBD232 : REAL ;
   DB9_DBD236 : REAL ;
   DB9_DBD240 : REAL ;
   DB9_DBD244 : REAL ;
   DB9_DBD248 : REAL ;
   DB9_DBD252 : REAL ;
   DB9_DBD256 : REAL ;
   DB9_DBD260 : REAL ;
   DB9_DBD264 : REAL ;
   DB9_DBD268 : REAL ;
  END_STRUCT ;	
BEGIN
   DB9_DBD20 := 3.000000e+00;
   DB9_DBD28 := 9.130859e-01;
   DB9_DBD32 := 2.725146e+01;
   DB9_DBD36 := 1.318359e-01;
   DB9_DBD40 := 5.444489e+01;
   DB9_DBD72 := 1.000000e+01;
   DB9_DBD76 := 1.000000e+01;
   DB9_DBD128 := 5.000000e+00;
END_DATA_BLOCK

DATA_BLOCK "Cage 24"	// DB 15
TITLE = CAGE 24 DATA BLOCK
AUTHOR : Milesi
VERSION : 0.1
  STRUCT
   HMI_Bit : STRUCT
    DB15_DBX0_0 : BOOL ;
    DB15_DBX0_1 : BOOL ;
    DB15_DBX0_2 : BOOL ;
    DB15_DBX0_3 : BOOL ;
    DB15_DBX0_4 : BOOL ;
    DB15_DBX0_5 : BOOL ;
    DB15_DBX0_6 : BOOL ;
    DB15_DBX0_7 : BOOL ;
    DB15_DBX1_0 : BOOL ;
    DB15_DBX1_1 : BOOL ;
    DB15_DBX1_2 : BOOL ;
    DB15_DBX1_3 : BOOL ;
    DB15_DBX1_4 : BOOL ;
    DB15_DBX1_5 : BOOL ;
    DB15_DBX1_6 : BOOL ;
    DB15_DBX1_7 : BOOL ;
   END_STRUCT ;
   DB15_DBW2 : INT ;	//Insertion 0=off 1=on from HMI
   DB15_DBW4 : INT ;	//Rotation 0=z 1=s from HMI
   DB15_DBW6 : S5TIME ;	//BCD constant
   DB15_DBW8 : INT ;
   DB15_DBW10 : INT ;
   DB15_DBW12 : INT ;	//Bobbins on read
   DB15_DBW14 : INT ;	//Bobbin 1 real diameter
   DB15_DBW16 : INT ;	//Bobbin 1 impulses for minute
   DB15_DBW18 : INT ;	//Number of wires inserted from HMI
   DB15_DBD20 : REAL ;	//Lay set from HMI
   DB15_DBD24 : REAL ;	//Lay set
   DB15_DBD28 : REAL ;	//Cable compacting % from HMI
   DB15_DBD32 : REAL ;
   DB15_DBD36 : REAL ;
   DB15_DBD40 : REAL ;
   DB15_DBD44 : REAL ;
   DB15_DBD48 : REAL ;
   DB15_DBD52 : REAL ;
   DB15_DBD56 : REAL ;
   DB15_DBD60 : REAL ;
   DB15_DBD64 : REAL ;	//Normal stop brake constant from HMI
   DB15_DBD68 : REAL ;	//Quick stop brake constant from HMI
   DB15_DBD72 : REAL ;	//Emergency stop brake constant from HMI
   DB15_DBD76 : REAL ;	//Missing power supply stop brake constant (copper) from HMI
   DB15_DBD80 : REAL ;	//Missing power supply stop brake reference
   DB15_DBD84 : REAL ;	//Aux1
   DB15_DBD88 : REAL ;
   DB15_DBD92 : REAL ;	//Jog rpm reference from HMI
   DB15_DBD96 : REAL ;	//Max linear speed
   DB15_DBD100 : REAL ;
   DB15_DBD104 : REAL ;	//Cable compacting costant
   DB15_DBD108 : REAL ;	//Rpm to HMI (ABS)
   DB15_DBD112 : REAL ;	//Diameter adjustment constant
   DB15_DBD116 : REAL ;	//Linear speed read adjusted by compact K
   DB15_DBD120 : REAL ;	//Max linear speed to start
   DB15_DBD124 : REAL ;
   DB15_DBD128 : REAL ;	//Bobbins wires pull set from HMI
   DB15_DBD132 : REAL ;
   DB15_DBD136 : REAL ;
   DB15_DBD140 : REAL ;
   DB15_DBD144 : REAL ;	//Piston's on-delay time outside cage from HMI
   DB15_DBD148 : REAL ;	//Brakes block open on-delay time from HMI
   DB15_DBD152 : REAL ;	//Piston's on-delay time inside cage from HMI
   DB15_DBD156 : REAL ;	//Air inlet on-delay time cage from HMI
   DB15_DBD160 : REAL ;
   DB15_DBD164 : REAL ;
   DB15_DBD168 : REAL ;
   DB15_DBD172 : REAL ;
   DB15_DBD176 : REAL ;
   DB15_DBD180 : REAL ;
   DB15_DBD184 : REAL ;
   DB15_DBD188 : REAL ;	//Motor rpm to HMI
   DB15_DBD192 : REAL ;	//Motor current to HMI
   DB15_DBD196 : REAL ;	//Motor voltage to HMI
   DB15_DBD200 : REAL ;	//Motor current for Brake control
   DB15_DBD204 : REAL ;	//Speed reference to drive
   DB15_DBD208 : REAL ;
   DB15_DBD212 : REAL ;
   DB15_DBD216 : REAL ;
   DB15_DBD220 : REAL ;
   DB15_DBD224 : REAL ;
   DB15_DBD228 : REAL ;
   DB15_DBD232 : REAL ;
   DB15_DBD236 : REAL ;
   DB15_DBD240 : REAL ;
   DB15_DBD244 : REAL ;
   DB15_DBD248 : REAL ;
   DB15_DBD252 : REAL ;
   DB15_DBD256 : REAL ;
   DB15_DBD260 : REAL ;	//Motor current Set point Amper
   DB15_DBD264 : REAL ;	//Motor current error
   DB15_DBD268 : REAL ;	//Brake control on current - proportional gain
   DB15_DBD272 : REAL ;	//Brake control on current - output
   DB15_DBD276 : REAL ;	//Motor current Set point 0-100% current from HMI
   DB15_DBD280 : REAL ;
   DB15_DBD284 : REAL ;
  END_STRUCT ;	
BEGIN
   DB15_DBW6 := S5T#0MS;
   DB15_DBW14 := 630;
   DB15_DBD20 := 1.000000e+02;
   DB15_DBD24 := 1.000000e+02;
   DB15_DBD28 := 1.000000e+02;
   DB15_DBD32 := 1.808533e+01;
   DB15_DBD36 := 2.438965e+00;
   DB15_DBD40 := 3.984375e+01;
   DB15_DBD64 := 1.000000e+01;
   DB15_DBD68 := 2.000000e+01;
   DB15_DBD72 := 4.000000e+01;
   DB15_DBD80 := 6.000000e+01;
   DB15_DBD84 := 6.000000e+01;
   DB15_DBD92 := 3.000000e+00;
   DB15_DBD96 := 6.000000e+01;
   DB15_DBD100 := 2.000000e+00;
   DB15_DBD104 := 8.000000e+00;
   DB15_DBD112 := 1.274000e+03;
   DB15_DBD116 := 5.000000e+00;
   DB15_DBD120 := 6.000000e+01;
   DB15_DBD124 := 1.000000e+00;
   DB15_DBD144 := 2.000000e+00;
   DB15_DBD152 := 2.000000e+00;
   DB15_DBD156 := 2.000000e+00;
   DB15_DBD200 := -0.000000e+00;
   DB15_DBD260 := 5.940000e+01;
   DB15_DBD264 := 5.940000e+01;
   DB15_DBD268 := 2.000000e+01;
   DB15_DBD272 := 1.188000e+03;
   DB15_DBD276 := 3.000000e+01;
END_DATA_BLOCK

DATA_BLOCK "Cage 24 preforming"	// DB 18
TITLE = CAGE 24 PREFORMING DATA BLOCK
AUTHOR : Milesi
VERSION : 0.1
  STRUCT
   HMI_Bit : STRUCT
    DB18_DBX0_0 : BOOL ;
    DB18_DBX0_1 : BOOL ;
    DB18_DBX0_2 : BOOL ;
    DB18_DBX0_3 : BOOL ;
    DB18_DBX0_4 : BOOL ;
    DB18_DBX0_5 : BOOL ;
    DB18_DBX0_6 : BOOL ;
    DB18_DBX0_7 : BOOL ;
    DB18_DBX1_0 : BOOL ;
    DB18_DBX1_1 : BOOL ;
    DB18_DBX1_2 : BOOL ;
    DB18_DBX1_3 : BOOL ;
    DB18_DBX1_4 : BOOL ;
    DB18_DBX1_5 : BOOL ;
    DB18_DBX1_6 : BOOL ;
    DB18_DBX1_7 : BOOL ;
   END_STRUCT ;
   DB18_DBW2 : INT ;	//Insertion 0=off 1=Z 2=S from HMI
   DB18_DBW4 : INT ;
   DB18_DBW6 : INT ;
   DB18_DBW8 : INT ;
   DB18_DBW10 : INT ;
   DB18_DBW12 : INT ;
   DB18_DBW14 : INT ;
   DB18_DBW16 : INT ;
   DB18_DBW18 : INT ;
   DB18_DBD20 : REAL ;	//Lay set from HMI
   DB18_DBD24 : REAL ;
   DB18_DBD28 : REAL ;
   DB18_DBD32 : REAL ;
   DB18_DBD36 : REAL ;
   DB18_DBD40 : REAL ;
   DB18_DBD44 : REAL ;
   DB18_DBD48 : REAL ;
   DB18_DBD52 : REAL ;
   DB18_DBD56 : REAL ;
   DB18_DBD60 : REAL ;
   DB18_DBD64 : REAL ;
   DB18_DBD68 : REAL ;
   DB18_DBD72 : REAL ;
   DB18_DBD76 : REAL ;
   DB18_DBD80 : REAL ;
   DB18_DBD84 : REAL ;
   DB18_DBD88 : REAL ;
   DB18_DBD92 : REAL ;
   DB18_DBD96 : REAL ;
   DB18_DBD100 : REAL ;
   DB18_DBD104 : REAL ;
   DB18_DBD108 : REAL ;	//Rpm to HMI (ABS)
   DB18_DBD112 : REAL ;
   DB18_DBD116 : REAL ;
   DB18_DBD120 : REAL ;
   DB18_DBD124 : REAL ;
   DB18_DBD128 : REAL ;
   DB18_DBD132 : REAL ;
   DB18_DBD136 : REAL ;
   DB18_DBD140 : REAL ;
   DB18_DBD144 : REAL ;
   DB18_DBD148 : REAL ;
   DB18_DBD152 : REAL ;
   DB18_DBD156 : REAL ;
   DB18_DBD160 : REAL ;
   DB18_DBD164 : REAL ;
   DB18_DBD168 : REAL ;
   DB18_DBD172 : REAL ;
   DB18_DBD176 : REAL ;
   DB18_DBD180 : REAL ;
   DB18_DBD184 : REAL ;
   DB18_DBD188 : REAL ;	//Motor rpm to HMI
   DB18_DBD192 : REAL ;	//Motor current to HMI
   DB18_DBD196 : REAL ;	//Motor voltage to HMI
   DB18_DBD200 : REAL ;
   DB18_DBD204 : REAL ;	//Speed reference to drive
   DB18_DBD208 : REAL ;
   DB18_DBD212 : REAL ;
   DB18_DBD216 : REAL ;
   DB18_DBD220 : REAL ;
   DB18_DBD224 : REAL ;
   DB18_DBD228 : REAL ;
   DB18_DBD232 : REAL ;
   DB18_DBD236 : REAL ;
   DB18_DBD240 : REAL ;
   DB18_DBD244 : REAL ;
   DB18_DBD248 : REAL ;
   DB18_DBD252 : REAL ;
   DB18_DBD256 : REAL ;
   DB18_DBD260 : REAL ;
   DB18_DBD264 : REAL ;
   DB18_DBD268 : REAL ;
   DB18_DBD272 : REAL ;
   DB18_DBD276 : REAL ;
  END_STRUCT ;	
BEGIN
   DB18_DBD20 := 5.000000e+02;
END_DATA_BLOCK

DATA_BLOCK "Cage 18"	// DB 20
TITLE = CAGE 18 DATA BLOCK
AUTHOR : Milesi
VERSION : 0.1
  STRUCT
   HMI_Bit : STRUCT
    DB20_DBX0_0 : BOOL ;
    DB13_DBX0_1 : BOOL ;
    DB20_DBX0_2 : BOOL ;
    DB20_DBX0_3 : BOOL ;
    DB20_DBX0_4 : BOOL ;
    DB20_DBX0_5 : BOOL ;
    DB20_DBX0_6 : BOOL ;
    DB20_DBX0_7 : BOOL ;
    DB20_DBX1_0 : BOOL ;
    DB20_DBX1_1 : BOOL ;
    DB20_DBX1_2 : BOOL ;
    DB20_DBX1_3 : BOOL ;
    DB20_DBX1_4 : BOOL ;
    DB20_DBX1_5 : BOOL ;
    DB20_DBX1_6 : BOOL ;
    DB20_DBX1_7 : BOOL ;
   END_STRUCT ;
   DB20_DBW2 : INT ;	//Insertion 0=off 1=on from HMI
   DB20_DBW4 : INT ;	//Rotation 0=z 1=s from HMI
   DB20_DBW6 : S5TIME ;	//BCD constant
   DB20_DBW8 : INT ;
   DB20_DBW10 : INT ;
   DB20_DBW12 : INT ;	//Bobbins on read
   DB20_DBW14 : INT ;	//Bobbin 1 real diameter
   DB20_DBW16 : INT ;	//Bobbin 1 impulses for minute
   DB20_DBW18 : INT ;	//Number of wires inserted from HMI
   DB20_DBD20 : REAL ;	//Lay set from HMI
   DB20_DBD24 : REAL ;	//Lay set
   DB20_DBD28 : REAL ;	//Cable compacting % from HMI
   DB20_DBD32 : REAL ;
   DB20_DBD36 : REAL ;
   DB20_DBD40 : REAL ;
   DB20_DBD44 : REAL ;
   DB20_DBD48 : REAL ;
   DB20_DBD52 : REAL ;
   DB20_DBD56 : REAL ;
   DB20_DBD60 : REAL ;
   DB20_DBD64 : REAL ;	//Normal stop brake constant from HMI
   DB20_DBD68 : REAL ;	//Quick stop brake constant from HMI
   DB20_DBD72 : REAL ;	//Emergency stop brake constant from HMI
   DB20_DBD76 : REAL ;	//Missing power supply stop brake constant (copper) from HMI
   DB20_DBD80 : REAL ;	//Missing power supply stop brake reference
   DB20_DBD84 : REAL ;	//Aux1
   DB20_DBD88 : REAL ;
   DB20_DBD92 : REAL ;	//Jog rpm reference from HMI
   DB20_DBD96 : REAL ;	//Max linear speed
   DB20_DBD100 : REAL ;
   DB20_DBD104 : REAL ;	//Cable compacting costant
   DB20_DBD108 : REAL ;	//Rpm to HMI (ABS)
   DB20_DBD112 : REAL ;	//Diameter adjustment constant
   DB20_DBD116 : REAL ;	//Linear speed read adjusted by compact K
   DB20_DBD120 : REAL ;	//Max linear speed to start
   DB20_DBD124 : REAL ;
   DB20_DBD128 : REAL ;	//Bobbins wires pull set from HMI
   DB20_DBD132 : REAL ;
   DB20_DBD136 : REAL ;
   DB20_DBD140 : REAL ;
   DB20_DBD144 : REAL ;	//Piston's on-delay time outside cage from HMI
   DB20_DBD148 : REAL ;	//Brakes block open on-delay time from HMI
   DB20_DBD152 : REAL ;	//Piston's on-delay time inside cage from HMI
   DB20_DBD156 : REAL ;	//Air inlet on-delay time cage from HMI
   DB20_DBD160 : REAL ;
   DB20_DBD164 : REAL ;
   DB20_DBD168 : REAL ;
   DB20_DBD172 : REAL ;
   DB20_DBD176 : REAL ;
   DB20_DBD180 : REAL ;
   DB20_DBD184 : REAL ;
   DB20_DBD188 : REAL ;	//Motor rpm to HMI
   DB20_DBD192 : REAL ;	//Motor current to HMI
   DB20_DBD196 : REAL ;	//Motor voltage to HMI
   DB20_DBD200 : REAL ;	//Motor current for Brake control
   DB20_DBD204 : REAL ;	//Speed reference to drive
   DB20_DBD208 : REAL ;
   DB20_DBD212 : REAL ;
   DB20_DBD216 : REAL ;
   DB20_DBD220 : REAL ;
   DB20_DBD224 : REAL ;
   DB20_DBD228 : REAL ;
   DB20_DBD232 : REAL ;
   DB20_DBD236 : REAL ;
   DB20_DBD240 : REAL ;
   DB20_DBD244 : REAL ;
   DB20_DBD248 : REAL ;
   DB20_DBD252 : REAL ;
   DB20_DBD256 : REAL ;
   DB20_DBD260 : REAL ;	//Motor current Set point current in amper
   DB20_DBD264 : REAL ;	//Motor current error
   DB20_DBD268 : REAL ;	//Brake control on current - proportional gain
   DB20_DBD272 : REAL ;	//Brake control on current - output
   DB20_DBD276 : REAL ;	//Motor current Set point 0-100% current from HMI
   DB20_DBD280 : REAL ;
   DB20_DBD284 : REAL ;
  END_STRUCT ;	
BEGIN
   DB20_DBW6 := S5T#0MS;
   DB20_DBW14 := 630;
   DB20_DBW18 := 18;
   DB20_DBD20 := 2.500000e+02;
   DB20_DBD24 := 2.500000e+02;
   DB20_DBD28 := 1.000000e+02;
   DB20_DBD32 := 1.808533e+01;
   DB20_DBD36 := 2.438965e+00;
   DB20_DBD40 := 3.984375e+01;
   DB20_DBD64 := 3.000000e+00;
   DB20_DBD68 := 3.000000e+01;
   DB20_DBD72 := 6.000000e+01;
   DB20_DBD80 := 6.000000e+01;
   DB20_DBD84 := 6.000000e+01;
   DB20_DBD92 := 3.000000e+00;
   DB20_DBD96 := 6.000000e+01;
   DB20_DBD100 := 2.000000e+00;
   DB20_DBD104 := 8.000000e+00;
   DB20_DBD112 := 1.274000e+03;
   DB20_DBD116 := 5.000000e+00;
   DB20_DBD120 := 6.000000e+01;
   DB20_DBD124 := 1.000000e+00;
   DB20_DBD128 := 1.500000e+01;
   DB20_DBD144 := 2.000000e+00;
   DB20_DBD152 := 2.000000e+00;
   DB20_DBD156 := 2.000000e+00;
   DB20_DBD200 := -0.000000e+00;
   DB20_DBD260 := 4.800000e+01;
   DB20_DBD264 := 4.800000e+01;
   DB20_DBD268 := 1.500000e+01;
   DB20_DBD272 := 7.200000e+02;
   DB20_DBD276 := 3.000000e+01;
END_DATA_BLOCK

DATA_BLOCK "Cage 18 preforming"	// DB 23
TITLE = CAGE 18 PREFORMING DATA BLOCK
AUTHOR : Milesi
VERSION : 0.1
  STRUCT
   HMI_Bit : STRUCT
    DB23_DBX0_0 : BOOL ;
    DB23_DBX0_1 : BOOL ;
    DB23_DBX0_2 : BOOL ;
    DB23_DBX0_3 : BOOL ;
    DB23_DBX0_4 : BOOL ;
    DB23_DBX0_5 : BOOL ;
    DB23_DBX0_6 : BOOL ;
    DB23_DBX0_7 : BOOL ;
    DB23_DBX1_0 : BOOL ;
    DB23_DBX1_1 : BOOL ;
    DB23_DBX1_2 : BOOL ;
    DB23_DBX1_3 : BOOL ;
    DB23_DBX1_4 : BOOL ;
    DB23_DBX1_5 : BOOL ;
    DB23_DBX1_6 : BOOL ;
    DB23_DBX1_7 : BOOL ;
   END_STRUCT ;
   DB23_DBW2 : INT ;	//Insertion 0=off 1=Z 2=S from HMI
   DB23_DBW4 : INT ;
   DB23_DBW6 : INT ;
   DB23_DBW8 : INT ;
   DB23_DBW10 : INT ;
   DB23_DBW12 : INT ;
   DB23_DBW14 : INT ;
   DB23_DBW16 : INT ;
   DB23_DBW18 : INT ;
   DB23_DBD20 : REAL ;	//Lay set from HMI
   DB23_DBD24 : REAL ;
   DB23_DBD28 : REAL ;
   DB23_DBD32 : REAL ;
   DB23_DBD36 : REAL ;
   DB23_DBD40 : REAL ;
   DB23_DBD44 : REAL ;
   DB23_DBD48 : REAL ;
   DB23_DBD52 : REAL ;
   DB23_DBD56 : REAL ;
   DB23_DBD60 : REAL ;
   DB23_DBD64 : REAL ;
   DB23_DBD68 : REAL ;
   DB23_DBD72 : REAL ;
   DB23_DBD76 : REAL ;
   DB23_DBD80 : REAL ;
   DB23_DBD84 : REAL ;
   DB23_DBD88 : REAL ;
   DB23_DBD92 : REAL ;
   DB23_DBD96 : REAL ;
   DB23_DBD100 : REAL ;
   DB23_DBD104 : REAL ;
   DB23_DBD108 : REAL ;	//Rpm to HMI (ABS)
   DB23_DBD112 : REAL ;
   DB23_DBD116 : REAL ;
   DB23_DBD120 : REAL ;
   DB23_DBD124 : REAL ;
   DB23_DBD128 : REAL ;
   DB23_DBD132 : REAL ;
   DB23_DBD136 : REAL ;
   DB23_DBD140 : REAL ;
   DB23_DBD144 : REAL ;
   DB23_DBD148 : REAL ;
   DB23_DBD152 : REAL ;
   DB23_DBD156 : REAL ;
   DB23_DBD160 : REAL ;
   DB23_DBD164 : REAL ;
   DB23_DBD168 : REAL ;
   DB23_DBD172 : REAL ;
   DB23_DBD176 : REAL ;
   DB23_DBD180 : REAL ;
   DB23_DBD184 : REAL ;
   DB23_DBD188 : REAL ;	//Motor rpm to HMI
   DB23_DBD192 : REAL ;	//Motor current to HMI
   DB23_DBD196 : REAL ;	//Motor voltage to HMI
   DB23_DBD200 : REAL ;
   DB23_DBD204 : REAL ;	//Speed reference to drive
   DB23_DBD208 : REAL ;
   DB23_DBD212 : REAL ;
   DB23_DBD216 : REAL ;
   DB23_DBD220 : REAL ;
   DB23_DBD224 : REAL ;
   DB23_DBD228 : REAL ;
   DB23_DBD232 : REAL ;
   DB23_DBD236 : REAL ;
   DB23_DBD240 : REAL ;
   DB23_DBD244 : REAL ;
   DB23_DBD248 : REAL ;
   DB23_DBD252 : REAL ;
   DB23_DBD256 : REAL ;
   DB23_DBD260 : REAL ;
   DB23_DBD264 : REAL ;
   DB23_DBD268 : REAL ;
   DB23_DBD272 : REAL ;
   DB23_DBD276 : REAL ;
  END_STRUCT ;	
BEGIN
   DB23_DBD20 := 2.788000e+03;
END_DATA_BLOCK

DATA_BLOCK "Cage 12"	// DB 25
TITLE = CAGE 12 DATA BLOCK
AUTHOR : Milesi
VERSION : 0.1
  STRUCT
   HMI_Bit : STRUCT
    DB25_DBX0_0 : BOOL ;
    DB25_DBX0_1 : BOOL ;
    DB25_DBX0_2 : BOOL ;
    DB25_DBX0_3 : BOOL ;
    DB25_DBX0_4 : BOOL ;
    DB25_DBX0_5 : BOOL ;
    DB25_DBX0_6 : BOOL ;
    DB25_DBX0_7 : BOOL ;
    DB25_DBX1_0 : BOOL ;
    DB25_DBX1_1 : BOOL ;
    DB25_DBX1_2 : BOOL ;
    DB25_DBX1_3 : BOOL ;
    DB25_DBX1_4 : BOOL ;
    DB25_DBX1_5 : BOOL ;
    DB25_DBX1_6 : BOOL ;
    DB25_DBX1_7 : BOOL ;
   END_STRUCT ;
   DB25_DBW2 : INT ;	//Insertion 0=off 1=on from HMI
   DB25_DBW4 : INT ;	//Rotation 0=z 1=s from HMI
   DB25_DBW6 : S5TIME ;	//BCD constant
   DB25_DBW8 : INT ;
   DB25_DBW10 : INT ;
   DB25_DBW12 : INT ;	//Bobbins on read
   DB25_DBW14 : INT ;	//Bobbin 1 real diameter
   DB25_DBW16 : INT ;	//Bobbin 1 impulses for minute
   DB25_DBW18 : INT ;	//Number of wires inserted from HMI
   DB25_DBD20 : REAL ;	//Lay set from HMI
   DB25_DBD24 : REAL ;	//Lay set
   DB25_DBD28 : REAL ;	//Cable compacting % from HMI
   DB25_DBD32 : REAL ;
   DB25_DBD36 : REAL ;
   DB25_DBD40 : REAL ;
   DB25_DBD44 : REAL ;
   DB25_DBD48 : REAL ;
   DB25_DBD52 : REAL ;
   DB25_DBD56 : REAL ;
   DB25_DBD60 : REAL ;
   DB25_DBD64 : REAL ;	//Normal stop brake constant from HMI
   DB25_DBD68 : REAL ;	//Quick stop brake constant from HMI
   DB25_DBD72 : REAL ;	//Emergency stop brake constant from HMI
   DB25_DBD76 : REAL ;	//Missing power supply stop brake constant (copper) from HMI
   DB25_DBD80 : REAL ;	//Missing power supply stop brake reference
   DB25_DBD84 : REAL ;	//Aux1
   DB25_DBD88 : REAL ;
   DB25_DBD92 : REAL ;	//Jog rpm reference from HMI
   DB25_DBD96 : REAL ;	//Max linear speed
   DB25_DBD100 : REAL ;
   DB25_DBD104 : REAL ;	//Cable compacting costant
   DB25_DBD108 : REAL ;	//Rpm to HMI (ABS)
   DB25_DBD112 : REAL ;	//Diameter adjustment constant
   DB25_DBD116 : REAL ;	//Linear speed read adjusted by compact K
   DB25_DBD120 : REAL ;	//Max linear speed to start
   DB25_DBD124 : REAL ;
   DB25_DBD128 : REAL ;	//Bobbins wires pull set from HMI
   DB25_DBD132 : REAL ;
   DB25_DBD136 : REAL ;
   DB25_DBD140 : REAL ;
   DB25_DBD144 : REAL ;	//Piston's on-delay time outside cage from HMI
   DB25_DBD148 : REAL ;	//Brakes block open on-delay time from HMI
   DB25_DBD152 : REAL ;	//Piston's on-delay time inside cage from HMI
   DB25_DBD156 : REAL ;	//Air inlet on-delay time cage from HMI
   DB25_DBD160 : REAL ;
   DB25_DBD164 : REAL ;
   DB25_DBD168 : REAL ;
   DB25_DBD172 : REAL ;
   DB25_DBD176 : REAL ;
   DB25_DBD180 : REAL ;
   DB25_DBD184 : REAL ;
   DB25_DBD188 : REAL ;	//Motor rpm to HMI
   DB25_DBD192 : REAL ;	//Motor current to HMI
   DB25_DBD196 : REAL ;	//Motor voltage to HMI
   DB25_DBD200 : REAL ;	//Motor current for Brake control
   DB25_DBD204 : REAL ;	//Speed reference to drive
   DB25_DBD208 : REAL ;
   DB25_DBD212 : REAL ;
   DB25_DBD216 : REAL ;
   DB25_DBD220 : REAL ;
   DB25_DBD224 : REAL ;
   DB25_DBD228 : REAL ;
   DB25_DBD232 : REAL ;
   DB25_DBD236 : REAL ;
   DB25_DBD240 : REAL ;
   DB25_DBD244 : REAL ;
   DB25_DBD248 : REAL ;
   DB25_DBD252 : REAL ;
   DB25_DBD256 : REAL ;
   DB20_DBD260 : REAL ;	//Motor current Set point current in amper
   DB20_DBD264 : REAL ;	//Motor current error
   DB20_DBD268 : REAL ;	//Brake control on current - proportional gain
   DB20_DBD272 : REAL ;	//Brake control on current - output
   DB20_DBD276 : REAL ;	//Motor current Set point 0-100% current from HMI
   DB20_DBD280 : REAL ;
   DB20_DBD284 : REAL ;
  END_STRUCT ;	
BEGIN
   DB25_DBW2 := 1;
   DB25_DBW4 := 1;
   DB25_DBW6 := S5T#0MS;
   DB25_DBW14 := 630;
   DB25_DBW18 := 12;
   DB25_DBD20 := 4.300000e+02;
   DB25_DBD24 := 4.300000e+02;
   DB25_DBD28 := 1.000000e+02;
   DB25_DBD32 := 1.808533e+01;
   DB25_DBD36 := 2.438965e+00;
   DB25_DBD40 := 3.984375e+01;
   DB25_DBD64 := 5.000000e+00;
   DB25_DBD68 := 3.300000e+01;
   DB25_DBD72 := 6.200000e+01;
   DB25_DBD80 := 6.000000e+01;
   DB25_DBD84 := 6.000000e+01;
   DB25_DBD92 := 3.000000e+00;
   DB25_DBD96 := 6.000000e+01;
   DB25_DBD100 := 2.000000e+00;
   DB25_DBD104 := 8.000000e+00;
   DB25_DBD112 := 1.274000e+03;
   DB25_DBD116 := 5.000000e+00;
   DB25_DBD120 := 6.000000e+01;
   DB25_DBD124 := 1.000000e+00;
   DB25_DBD128 := 2.000000e+01;
   DB25_DBD144 := 2.000000e+00;
   DB25_DBD152 := 2.000000e+00;
   DB25_DBD156 := 2.000000e+00;
   DB20_DBD260 := 4.080000e+01;
   DB20_DBD264 := 4.080000e+01;
   DB20_DBD268 := 1.500000e+01;
   DB20_DBD272 := 6.120000e+02;
   DB20_DBD276 := 3.000000e+01;
END_DATA_BLOCK

DATA_BLOCK "Cage 12 preforming"	// DB 28
TITLE = CAGE 12 PREFORMING DATA BLOCK
AUTHOR : Milesi
VERSION : 0.1
  STRUCT
   HMI_Bit : STRUCT
    DB28_DBX0_0 : BOOL ;
    DB28_DBX0_1 : BOOL ;
    DB28_DBX0_2 : BOOL ;
    DB28_DBX0_3 : BOOL ;
    DB28_DBX0_4 : BOOL ;
    DB28_DBX0_5 : BOOL ;
    DB28_DBX0_6 : BOOL ;
    DB28_DBX0_7 : BOOL ;
    DB28_DBX1_0 : BOOL ;
    DB28_DBX1_1 : BOOL ;
    DB28_DBX1_2 : BOOL ;
    DB28_DBX1_3 : BOOL ;
    DB28_DBX1_4 : BOOL ;
    DB28_DBX1_5 : BOOL ;
    DB28_DBX1_6 : BOOL ;
    DB28_DBX1_7 : BOOL ;
   END_STRUCT ;
   DB28_DBW2 : INT ;	//Insertion 0=off 1=Z 2=S from HMI
   DB28_DBW4 : INT ;
   DB28_DBW6 : S5TIME ;	//BCD constant
   DB28_DBW8 : INT ;
   DB28_DBW10 : INT ;
   DB28_DBW12 : INT ;
   DB28_DBW14 : INT ;
   DB28_DBW16 : INT ;
   DB28_DBW18 : INT ;
   DB28_DBD20 : REAL ;	//Lay set from HMI
   DB28_DBD24 : REAL ;
   DB28_DBD28 : REAL ;
   DB28_DBD32 : REAL ;
   DB28_DBD36 : REAL ;
   DB28_DBD40 : REAL ;
   DB28_DBD44 : REAL ;
   DB28_DBD48 : REAL ;
   DB28_DBD52 : REAL ;
   DB28_DBD56 : REAL ;
   DB28_DBD60 : REAL ;
   DB28_DBD64 : REAL ;
   DB28_DBD68 : REAL ;
   DB28_DBD72 : REAL ;
   DB28_DBD76 : REAL ;
   DB28_DBD80 : REAL ;
   DB28_DBD84 : REAL ;
   DB28_DBD88 : REAL ;
   DB28_DBD92 : REAL ;
   DB28_DBD96 : REAL ;
   DB28_DBD100 : REAL ;
   DB28_DBD104 : REAL ;
   DB28_DBD108 : REAL ;	//Rpm to HMI (ABS)
   DB28_DBD112 : REAL ;
   DB28_DBD116 : REAL ;
   DB28_DBD120 : REAL ;
   DB28_DBD124 : REAL ;
   DB28_DBD128 : REAL ;
   DB28_DBD132 : REAL ;
   DB28_DBD136 : REAL ;
   DB28_DBD140 : REAL ;
   DB28_DBD144 : REAL ;
   DB28_DBD148 : REAL ;
   DB28_DBD152 : REAL ;
   DB28_DBD156 : REAL ;
   DB28_DBD160 : REAL ;
   DB28_DBD164 : REAL ;
   DB28_DBD168 : REAL ;
   DB28_DBD172 : REAL ;
   DB28_DBD176 : REAL ;
   DB28_DBD180 : REAL ;
   DB28_DBD184 : REAL ;
   DB28_DBD188 : REAL ;	//Motor rpm to HMI
   DB28_DBD192 : REAL ;	//Motor current to HMI
   DB28_DBD196 : REAL ;	//Motor voltage to HMI
   DB28_DBD200 : REAL ;
   DB28_DBD204 : REAL ;	//Speed reference to drive
   DB28_DBD208 : REAL ;
   DB28_DBD212 : REAL ;
   DB28_DBD216 : REAL ;
   DB28_DBD220 : REAL ;
   DB28_DBD224 : REAL ;
   DB28_DBD228 : REAL ;
   DB28_DBD232 : REAL ;
   DB28_DBD236 : REAL ;
   DB28_DBD240 : REAL ;
   DB28_DBD244 : REAL ;
   DB28_DBD248 : REAL ;
   DB28_DBD252 : REAL ;
   DB28_DBD256 : REAL ;
   DB28_DBD260 : REAL ;
   DB28_DBD264 : REAL ;
   DB28_DBD268 : REAL ;
   DB28_DBD272 : REAL ;
   DB28_DBD276 : REAL ;
  END_STRUCT ;	
BEGIN
   DB28_DBD20 := 2.788000e+03;
END_DATA_BLOCK

DATA_BLOCK "Cage 6"	// DB 30
TITLE = CAGE 6 DATA BLOCK
AUTHOR : Milesi
VERSION : 0.1
  STRUCT
   HMI_Bit : STRUCT
    DB30_DBX0_0 : BOOL ;
    DB30_DBX0_1 : BOOL ;
    DB30_DBX0_2 : BOOL ;
    DB30_DBX0_3 : BOOL ;
    DB30_DBX0_4 : BOOL ;
    DB30_DBX0_5 : BOOL ;
    DB30_DBX0_6 : BOOL ;
    DB30_DBX0_7 : BOOL ;
    DB30_DBX1_0 : BOOL ;
    DB30_DBX1_1 : BOOL ;
    DB30_DBX1_2 : BOOL ;
    DB30_DBX1_3 : BOOL ;
    DB30_DBX1_4 : BOOL ;
    DB30_DBX1_5 : BOOL ;
    DB30_DBX1_6 : BOOL ;
    DB30_DBX1_7 : BOOL ;
   END_STRUCT ;
   DB30_DBW2 : INT ;	//Insertion 0=off 1=on from HMI
   DB30_DBW4 : INT ;	//Rotation 0=z 1=s from HMI
   DB30_DBW6 : S5TIME ;	//BCD constant
   DB30_DBW8 : INT ;
   DB30_DBW10 : INT ;
   DB30_DBW12 : INT ;	//Bobbins on read
   DB30_DBW14 : INT ;	//Bobbin 1 real diameter
   DB30_DBW16 : INT ;	//Bobbin 1 impulses for minute
   DB30_DBW18 : INT ;	//Number of wires inserted from HMI
   DB30_DBD20 : REAL ;	//Lay set from HMI
   DB30_DBD24 : REAL ;	//Lay set
   DB30_DBD28 : REAL ;	//Cable compacting % from HMI
   DB30_DBD32 : REAL ;
   DB30_DBD36 : REAL ;
   DB30_DBD40 : REAL ;
   DB30_DBD44 : REAL ;
   DB30_DBD48 : REAL ;
   DB30_DBD52 : REAL ;
   DB30_DBD56 : REAL ;
   DB30_DBD60 : REAL ;
   DB30_DBD64 : REAL ;	//Normal stop brake constant from HMI
   DB30_DBD68 : REAL ;	//Quick stop brake constant from HMI
   DB30_DBD72 : REAL ;	//Emergency stop brake constant from HMI
   DB30_DBD76 : REAL ;	//Missing power supply stop brake constant (copper) from HMI
   DB30_DBD80 : REAL ;	//Missing power supply stop brake reference
   DB30_DBD84 : REAL ;	//Aux1
   DB30_DBD88 : REAL ;
   DB30_DBD92 : REAL ;	//Jog rpm reference from HMI
   DB30_DBD96 : REAL ;	//Max linear speed
   DB30_DBD100 : REAL ;
   DB30_DBD104 : REAL ;	//Cable compacting costant
   DB30_DBD108 : REAL ;	//Rpm to HMI (ABS)
   DB30_DBD112 : REAL ;	//Diameter adjustment constant
   DB30_DBD116 : REAL ;	//Linear speed read adjusted by compact K
   DB30_DBD120 : REAL ;	//Max linear speed to start
   DB30_DBD124 : REAL ;
   DB30_DBD128 : REAL ;	//Bobbins wires pull set from HMI
   DB30_DBD132 : REAL ;
   DB30_DBD136 : REAL ;
   DB30_DBD140 : REAL ;
   DB30_DBD144 : REAL ;	//Piston's on-delay time outside cage from HMI
   DB30_DBD148 : REAL ;	//Brakes block open on-delay time from HMI
   DB30_DBD152 : REAL ;	//Piston's on-delay time inside cage from HMI
   DB30_DBD156 : REAL ;	//Air inlet on-delay time cage from HMI
   DB30_DBD160 : REAL ;
   DB30_DBD164 : REAL ;
   DB30_DBD168 : REAL ;
   DB30_DBD172 : REAL ;
   DB30_DBD176 : REAL ;
   DB30_DBD180 : REAL ;
   DB30_DBD184 : REAL ;
   DB30_DBD188 : REAL ;	//Motor rpm to HMI
   DB30_DBD192 : REAL ;	//Motor current to HMI
   DB30_DBD196 : REAL ;	//Motor voltage to HMI
   DB30_DBD200 : REAL ;	//Motor current for Brake control
   DB30_DBD204 : REAL ;	//Speed reference to drive
   DB30_DBD208 : REAL ;
   DB30_DBD212 : REAL ;
   DB30_DBD216 : REAL ;
   DB30_DBD220 : REAL ;
   DB30_DBD224 : REAL ;
   DB30_DBD228 : REAL ;
   DB30_DBD232 : REAL ;
   DB30_DBD236 : REAL ;
   DB30_DBD240 : REAL ;
   DB30_DBD244 : REAL ;
   DB30_DBD248 : REAL ;
   DB30_DBD252 : REAL ;
   DB30_DBD256 : REAL ;
   DB20_DBD260 : REAL ;	//Motor current Set point current in amper
   DB20_DBD264 : REAL ;	//Motor current error
   DB20_DBD268 : REAL ;	//Brake control on current - proportional gain
   DB20_DBD272 : REAL ;	//Brake control on current - output
   DB20_DBD276 : REAL ;	//Motor current Set point 0-100% current from HMI
   DB20_DBD280 : REAL ;
   DB20_DBD284 : REAL ;
  END_STRUCT ;	
BEGIN
   DB30_DBW2 := 1;
   DB30_DBW6 := S5T#0MS;
   DB30_DBW14 := 400;
   DB30_DBW18 := 6;
   DB30_DBD20 := 3.170000e+02;
   DB30_DBD24 := 3.170000e+02;
   DB30_DBD28 := 5.613708e+01;
   DB30_DBD32 := 9.637695e+00;
   DB30_DBD36 := 8.997803e+00;
   DB30_DBD40 := 1.401764e+01;
   DB30_DBD64 := 1.000000e+01;
   DB30_DBD68 := 3.000000e+01;
   DB30_DBD72 := 6.000000e+01;
   DB30_DBD80 := 5.000000e+01;
   DB30_DBD84 := 5.000000e+01;
   DB30_DBD92 := 3.000000e+00;
   DB30_DBD96 := 6.000000e+01;
   DB30_DBD100 := 2.000000e+00;
   DB30_DBD104 := 8.000000e+00;
   DB30_DBD112 := 1.274000e+03;
   DB30_DBD120 := 6.000000e+01;
   DB30_DBD124 := 1.000000e+00;
   DB30_DBD128 := 1.100000e+01;
   DB30_DBD144 := 2.000000e+00;
   DB30_DBD152 := 2.000000e+00;
   DB30_DBD156 := 2.000000e+00;
   DB30_DBD200 := -0.000000e+00;
   DB20_DBD260 := 3.000000e+01;
   DB20_DBD264 := 3.000000e+01;
   DB20_DBD268 := 4.000000e+01;
   DB20_DBD272 := 1.200000e+03;
   DB20_DBD276 := 3.000000e+01;
END_DATA_BLOCK

DATA_BLOCK "Pay-off 630"	// DB 35
TITLE = PAY-OFF 630 DATA BLOCK
AUTHOR : Milesi
VERSION : 0.1
  STRUCT
   HMI_Bit : STRUCT
    DB35_DBX0_0 : BOOL ;
    DB35_DBX0_1 : BOOL ;
    DB35_DBX0_2 : BOOL ;
    DB35_DBX0_3 : BOOL ;
    DB35_DBX0_4 : BOOL ;
    DB35_DBX0_5 : BOOL ;
    DB35_DBX0_6 : BOOL ;
    DB35_DBX0_7 : BOOL ;
    DB35_DBX1_0 : BOOL ;	//Insertion from HMI (0=off 1=on)
    DB35_DBX1_1 : BOOL ;	//Wire break control insertion from HMI (0=off 1= on)
    DB35_DBX1_2 : BOOL ;
    DB35_DBX1_3 : BOOL ;
    DB35_DBX1_4 : BOOL ;
    DB35_DBX1_5 : BOOL ;
    DB35_DBX1_6 : BOOL ;
    DB35_DBX1_7 : BOOL ;	//Insertion on to HMI
   END_STRUCT ;
   DB35_DBW2 : INT ;
   DB35_DBW4 : INT ;
   DB35_DBW6 : S5TIME ;	//BCD constant
   DB35_DBW8 : INT ;
   DB35_DBW10 : INT ;
   DB35_DBW12 : INT ;
   DB35_DBW14 : INT ;	//Bobbin real diameter
   DB35_DBW16 : INT ;	//Bobbin impulses for minute
   DB35_DBW18 : INT ;
   DB35_DBD20 : REAL ;	//Bobbin pull set from HMI
   DB35_DBD24 : REAL ;
   DB35_DBD28 : REAL ;
   DB35_DBD32 : REAL ;
   DB35_DBD36 : REAL ;
   DB35_DBD40 : REAL ;
   DB35_DBD44 : REAL ;
   DB35_DBD48 : REAL ;
   DB35_DBD52 : REAL ;
   DB35_DBD56 : REAL ;
   DB35_DBD60 : REAL ;
   DB35_DBD64 : REAL ;
   DB35_DBD68 : REAL ;
   DB35_DBD72 : REAL ;
   DB35_DBD76 : REAL ;
   DB35_DBD80 : REAL ;
   DB35_DBD84 : REAL ;
   DB35_DBD88 : REAL ;
   DB35_DBD92 : REAL ;
   DB35_DBD96 : REAL ;
   DB35_DBD100 : REAL ;
   DB35_DBD104 : REAL ;
   DB35_DBD108 : REAL ;
   DB35_DBD112 : REAL ;
   DB35_DBD116 : REAL ;
   DB35_DBD120 : REAL ;
   DB35_DBD124 : REAL ;
   DB35_DBD128 : REAL ;
   DB35_DBD132 : REAL ;
   DB35_DBD136 : REAL ;
   DB35_DBD140 : REAL ;
   DB35_DBD144 : REAL ;
   DB35_DBD148 : REAL ;
   DB35_DBD152 : REAL ;
   DB35_DBD156 : REAL ;
   DB35_DBD160 : REAL ;
   DB35_DBD164 : REAL ;
   DB35_DBD168 : REAL ;
   DB35_DBD172 : REAL ;
   DB35_DBD176 : REAL ;
   DB35_DBD180 : REAL ;
   DB35_DBD184 : REAL ;
   DB35_DBD188 : REAL ;
   DB35_DBD192 : REAL ;
   DB35_DBD196 : REAL ;
  END_STRUCT ;	
BEGIN
   HMI_Bit.DB35_DBX1_0 := TRUE;
   HMI_Bit.DB35_DBX1_7 := TRUE;
   DB35_DBW6 := S5T#0MS;
   DB35_DBW10 := 465;
   DB35_DBW14 := 400;
   DB35_DBD20 := 1.000000e+01;
   DB35_DBD112 := 1.274000e+03;
END_DATA_BLOCK

DATA_BLOCK "Metercounter"	// DB 41
TITLE = METERCOUNTER DATA BLOCK
AUTHOR : Milesi
VERSION : 0.1
  STRUCT
   HMI_Bit : STRUCT
    DB41_DBX0_0 : BOOL ;
    DB41_DBX0_1 : BOOL ;
    DB41_DBX0_2 : BOOL ;
    DB41_DBX0_3 : BOOL ;
    DB41_DBX0_4 : BOOL ;
    DB41_DBX0_5 : BOOL ;
    DB41_DBX0_6 : BOOL ;
    DB41_DBX0_7 : BOOL ;
    DB41_DBX1_0 : BOOL ;	//Actual lenght reset
    DB41_DBX1_1 : BOOL ;	//Actual total lenght reset
    DB41_DBX1_2 : BOOL ;
    DB41_DBX1_3 : BOOL ;
    DB41_DBX1_4 : BOOL ;
    DB41_DBX1_5 : BOOL ;
    DB41_DBX1_6 : BOOL ;
    DB41_DBX1_7 : BOOL ;
   END_STRUCT ;
   DB41_DBW2 : INT ;
   DB41_DBW4 : INT ;
   DB41_DBW6 : INT ;
   DB41_DBW8 : INT ;
   DB41_DBW10 : INT ;
   DB41_DBW12 : INT ;
   DB41_DBW14 : INT ;
   DB41_DBW16 : INT ;
   DB41_DBW18 : INT ;
   DB41_DBD20 : REAL ;
   DB41_DBD24 : REAL ;
   DB41_DBD28 : REAL ;
   DB41_DBD32 : REAL ;	//Lenght set from HMI
   DB41_DBD36 : REAL ;	//Deceleration lenght set from HMI
   DB41_DBD40 : REAL ;	//Actual total lenght
   DB41_DBD44 : REAL ;	//Actual lenght
   DB41_DBD48 : REAL ;	//Constant set from HMI
   DB41_DBD52 : REAL ;	//Lenght to make
   DB41_DBD56 : REAL ;
   DB41_DBD60 : REAL ;
   DB41_DBD64 : REAL ;
   DB41_DBD68 : REAL ;
   DB41_DBD72 : REAL ;	//Lenght increase (m)
   DB41_DBD76 : REAL ;
   DB41_DBD80 : REAL ;
   DB41_DBD84 : REAL ;
   DB41_DBD88 : REAL ;
   DB41_DBD92 : REAL ;
   DB41_DBD96 : REAL ;
   DB41_DBD100 : REAL ;
   DB41_DBD104 : REAL ;
   DB41_DBD108 : REAL ;
   DB41_DBD111 : REAL ;
   DB41_DBD116 : REAL ;
   DB41_DBD120 : REAL ;
   DB41_DBD124 : REAL ;
   DB41_DBD128 : REAL ;
   DB41_DBD132 : DINT ;	//Encoder counter hold
   DB41_DBD136 : REAL ;
   DB41_DBD140 : REAL ;
   DB41_DBD144 : REAL ;
   DB41_DBD148 : REAL ;
   DB41_DBD152 : REAL ;
   DB41_DBD156 : REAL ;
   DB41_DBD160 : REAL ;
   DB41_DBD164 : REAL ;
   DB41_DBD168 : REAL ;
   DB41_DBD172 : REAL ;
   DB41_DBD176 : REAL ;
   DB41_DBD180 : REAL ;
   DB41_DBD184 : REAL ;
   DB41_DBD188 : REAL ;
   DB41_DBD192 : REAL ;
   DB41_DBD196 : REAL ;
  END_STRUCT ;	
BEGIN
   DB41_DBD32 := 2.000000e+03;
   DB41_DBD36 := 3.000000e+01;
   DB41_DBD40 := 3.119794e+03;
   DB41_DBD44 := 1.118888e+03;
   DB41_DBD48 := 1.000000e+00;
   DB41_DBD52 := 8.811119e+02;
   DB41_DBD104 := 2.527000e+03;
   DB41_DBD111 := 1.106199e+03;
   DB41_DBD116 := -1.268872e+01;
   DB41_DBD132 := L#13766154;
END_DATA_BLOCK

DATA_BLOCK "Line"	// DB 55
TITLE = LINE DATA BLOCK
AUTHOR : Milesi
VERSION : 0.1
  STRUCT
   HMI_Bit : STRUCT
    DB55_DBX0_0 : BOOL ;
    DB55_DBX0_1 : BOOL ;
    DB55_DBX0_2 : BOOL ;
    DB55_DBX0_3 : BOOL ;
    DB55_DBX0_4 : BOOL ;
    DB55_DBX0_5 : BOOL ;
    DB55_DBX0_6 : BOOL ;
    DB55_DBX0_7 : BOOL ;
    DB55_DBX1_0 : BOOL ;
    DB55_DBX1_1 : BOOL ;	//Material from HMI (0=copper/steel; 1=alluminium)
    DB55_DBX1_2 : BOOL ;	//
    DB55_DBX1_3 : BOOL ;	//
    DB55_DBX1_4 : BOOL ;	//
    DB55_DBX1_5 : BOOL ;	//
    DB55_DBX1_6 : BOOL ;	//
    DB55_DBX1_7 : BOOL ;	//
   END_STRUCT ;
   DB55_DBW2 : INT ;	//Production from HMI (0=straight sect; 1=preformed sect; 2 round; 3 armoured)
   DB55_DBW4 : INT ;
   DB55_DBW6 : INT ;
   DB55_DBW8 : INT ;
   DB55_DBW10 : INT ;
   DB55_DBW12 : INT ;
   DB55_DBW14 : INT ;
   DB55_DBW16 : INT ;
   DB55_DBW18 : INT ;
   DB55_DBD20 : REAL ;	//Second counter
   DB55_DBD24 : REAL ;	//Hour counter
   DB55_DBD28 : REAL ;	//Linear speed set from HMI
   DB55_DBD32 : REAL ;	//Maximum linear speed set from HMI
   DB55_DBD36 : REAL ;	//Line jog linear speed set from HMI
   DB55_DBD40 : REAL ;	//Linear speed limit to HMI
   DB55_DBD44 : REAL ;	//Line ramp up-down time from HMI
   DB55_DBD48 : REAL ;	//Linear speed reference
   DB55_DBD52 : REAL ;	//Capstan pinion gear grease hour counter
   DB55_DBD56 : REAL ;	//Cable diameter set from HMI
   DB55_DBD60 : REAL ;	//Line linear speed reference
   DB55_DBD64 : REAL ;	//Line stop ramp down time
   DB55_DBD68 : REAL ;	//Linear speed read (m/min)
   DB55_DBD72 : REAL ;	//Line linear speed to start
   DB55_DBD76 : REAL ;	//Line linear speed increase
   DB55_DBD80 : REAL ;	//Line linear speed to start + Line linear speed increase
   DB55_DBD84 : REAL ;	//Final line linear speed
   DB55_DBD88 : REAL ;	//Master cage rpm
   DB55_DBD92 : REAL ;	//Wire diameter set from HMI
   DB55_DBD96 : REAL ;	//Ramp output REAL 10000
   DB55_DBD100 : DINT ;	//Ramp output DINT 10000
   DB55_DBD104 : REAL ;	//Ramp output DWORD 100
   DB55_DBD108 : REAL ;
   DB55_DBD112 : REAL ;
   DB55_DBD116 : REAL ;
   DB55_DBD120 : REAL ;
   DB55_DBD124 : REAL ;
   DB55_DBD128 : REAL ;
   DB55_DBD132 : REAL ;	//Line run on-delay time from HMI
   DB55_DBD136 : REAL ;	//Breaking control on-delay time from HMI
   DB55_DBD140 : REAL ;	//Brakes-oil control on-delay time from HMI
   DB55_DBD144 : REAL ;	//Guards motor blower off-delay time from HMI
   DB55_DBD148 : REAL ;
   DB55_DBD152 : REAL ;
   DB55_DBD156 : REAL ;	//Increase mm from HMI
   DB55_DBD160 : REAL ;	//Increase time set from HMI
   DB55_DBD164 : REAL ;	//Number of steps sum for linear speed increasing
   DB55_DBD168 : REAL ;	//Linear speed increase actual time
   DB55_DBD172 : REAL ;	//Diameter of start
   DB55_DBD176 : REAL ;	//Calculate step REAL
   DB55_DBD180 : REAL ;
   DB55_DBD184 : REAL ;	//Step to make -1
   DB55_DBD188 : REAL ;	//Diameter next step
   DB55_DBD192 : REAL ;	//Master bobbin actual diameter
   DB55_DBD196 : REAL ;	//Linear speed increase single step
   DB55_DBD200 : REAL ;	//Missing supply brake control refresh time set from HMI
  END_STRUCT ;	
BEGIN
   HMI_Bit.DB55_DBX1_0 := TRUE;
   HMI_Bit.DB55_DBX1_1 := TRUE;
   DB55_DBW2 := 1;
   DB55_DBD20 := 1.300000e+02;
   DB55_DBD24 := 8.000000e+00;
   DB55_DBD28 := 5.000000e+00;
   DB55_DBD32 := 6.000000e+01;
   DB55_DBD36 := 3.000000e+00;
   DB55_DBD40 := 4.000000e+01;
   DB55_DBD44 := 1.200000e+02;
   DB55_DBD48 := 5.000000e+00;
   DB55_DBD52 := 2.700000e+01;
   DB55_DBD56 := 2.700000e+01;
   DB55_DBD64 := 1.200000e+01;
   DB55_DBD72 := 6.000000e+01;
   DB55_DBD80 := 6.000000e+01;
   DB55_DBD84 := 8.333334e+02;
   DB55_DBD92 := 2.960000e+00;
   DB55_DBD120 := 6.023804e+00;
   DB55_DBD132 := 2.000000e+00;
   DB55_DBD136 := 8.000000e+00;
   DB55_DBD140 := 5.000000e+00;
   DB55_DBD144 := 2.000000e+01;
   DB55_DBD156 := 1.000000e+01;
   DB55_DBD160 := 6.000000e+01;
   DB55_DBD172 := 6.300000e+02;
   DB55_DBD176 := 2.750000e+01;
   DB55_DBD184 := 2.650000e+01;
   DB55_DBD188 := 6.200000e+02;
   DB55_DBD192 := 4.000000e+02;
   DB55_DBD196 := -7.547170e-01;
END_DATA_BLOCK

